// BODAS_RC18_12_40/Application/02 EasyConfig/DSM_easyConfig/Structure/DFC_bds_NoDeb0x80e2
{attribute 'external_name' := 'cmp_rts_DFC_bds_NoDeb0x80e2'}
TYPE DFC_bds_NoDeb0x80e2 : STRUCT
        DTC            : UDINT := 16#80E200;
        DFCid          : UINT  := 28;
        debounceMethod : USINT := TIME_IN_ROW;
    END_STRUCT
END_TYPE

// BODAS_RC18_12_40/Application/02 EasyConfig/DSM_easyConfig/Structure/DFC_bds_NoDeb0x80e3
{attribute 'external_name' := 'cmp_rts_DFC_bds_NoDeb0x80e3'}
TYPE DFC_bds_NoDeb0x80e3 : STRUCT
        DTC            : UDINT := 16#80E300;
        DFCid          : UINT  := 29;
        debounceMethod : USINT := TIME_IN_ROW;
    END_STRUCT
END_TYPE

// BODAS_RC18_12_40/Application/02 EasyConfig/DSM_easyConfig/Structure/DFC_bds_NoDeb0x80e4
{attribute 'external_name' := 'cmp_rts_DFC_bds_NoDeb0x80e4'}
TYPE DFC_bds_NoDeb0x80e4 : STRUCT
        DTC            : UDINT := 16#80E400;
        DFCid          : UINT  := 30;
        debounceMethod : USINT := TIME_IN_ROW;
    END_STRUCT
END_TYPE

// BODAS_RC18_12_40/Application/02 EasyConfig/DSM_easyConfig/Structure/DFC_bds_NoDeb0x80e5
{attribute 'external_name' := 'cmp_rts_DFC_bds_NoDeb0x80e5'}
TYPE DFC_bds_NoDeb0x80e5 : STRUCT
        DTC            : UDINT := 16#80E500;
        DFCid          : UINT  := 31;
        debounceMethod : USINT := TIME_IN_ROW;
    END_STRUCT
END_TYPE

// BODAS_RC18_12_40/Application/02 EasyConfig/DSM_easyConfig/Structure/DFC_bds_NoDeb0x80e6
{attribute 'external_name' := 'cmp_rts_DFC_bds_NoDeb0x80e6'}
TYPE DFC_bds_NoDeb0x80e6 : STRUCT
        DTC            : UDINT := 16#80E600;
        DFCid          : UINT  := 32;
        debounceMethod : USINT := TIME_IN_ROW;
    END_STRUCT
END_TYPE

// BODAS_RC18_12_40/Application/02 EasyConfig/DSM_easyConfig/Structure/DFC_bds_NoDeb0x80e7
{attribute 'external_name' := 'cmp_rts_DFC_bds_NoDeb0x80e7'}
TYPE DFC_bds_NoDeb0x80e7 : STRUCT
        DTC            : UDINT := 16#80E700;
        DFCid          : UINT  := 33;
        debounceMethod : USINT := TIME_IN_ROW;
    END_STRUCT
END_TYPE

// BODAS_RC18_12_40/Application/02 EasyConfig/DSM_easyConfig/Structure/DFC_bds_NoDeb0x80e8
{attribute 'external_name' := 'cmp_rts_DFC_bds_NoDeb0x80e8'}
TYPE DFC_bds_NoDeb0x80e8 : STRUCT
        DTC            : UDINT := 16#80E800;
        DFCid          : UINT  := 34;
        debounceMethod : USINT := TIME_IN_ROW;
    END_STRUCT
END_TYPE

// BODAS_RC18_12_40/Application/02 EasyConfig/DSM_easyConfig/Structure/DFC_bds_NoDeb0x80e9
{attribute 'external_name' := 'cmp_rts_DFC_bds_NoDeb0x80e9'}
TYPE DFC_bds_NoDeb0x80e9 : STRUCT
        DTC            : UDINT := 16#80E900;
        DFCid          : UINT  := 35;
        debounceMethod : USINT := TIME_IN_ROW;
    END_STRUCT
END_TYPE

// BODAS_RC18_12_40/Application/02 EasyConfig/DSM_easyConfig/Structure/DFC_bds_NoDeb0x80ea
{attribute 'external_name' := 'cmp_rts_DFC_bds_NoDeb0x80ea'}
TYPE DFC_bds_NoDeb0x80ea : STRUCT
        DTC            : UDINT := 16#80EA00;
        DFCid          : UINT  := 36;
        debounceMethod : USINT := TIME_IN_ROW;
    END_STRUCT
END_TYPE

// BODAS_RC18_12_40/Application/02 EasyConfig/DSM_easyConfig/Structure/DFC_bds_NoDeb0x80eb
{attribute 'external_name' := 'cmp_rts_DFC_bds_NoDeb0x80eb'}
TYPE DFC_bds_NoDeb0x80eb : STRUCT
        DTC            : UDINT := 16#80EB00;
        DFCid          : UINT  := 37;
        debounceMethod : USINT := TIME_IN_ROW;
    END_STRUCT
END_TYPE

// BODAS_RC18_12_40/Application/02 EasyConfig/DSM_easyConfig/Structure/DFC_bds_NoDeb0x80ec
{attribute 'external_name' := 'cmp_rts_DFC_bds_NoDeb0x80ec'}
TYPE DFC_bds_NoDeb0x80ec : STRUCT
        DTC            : UDINT := 16#80EC00;
        DFCid          : UINT  := 38;
        debounceMethod : USINT := TIME_IN_ROW;
    END_STRUCT
END_TYPE

// BODAS_RC18_12_40/Application/02 EasyConfig/DSM_easyConfig/Structure/DFC_bds_NoDeb0x80ed
{attribute 'external_name' := 'cmp_rts_DFC_bds_NoDeb0x80ed'}
TYPE DFC_bds_NoDeb0x80ed : STRUCT
        DTC            : UDINT := 16#80ED00;
        DFCid          : UINT  := 39;
        debounceMethod : USINT := TIME_IN_ROW;
    END_STRUCT
END_TYPE

// BODAS_RC18_12_40/Application/02 EasyConfig/DSM_easyConfig/Structure/DFC_bds_NoDeb0x80ee
{attribute 'external_name' := 'cmp_rts_DFC_bds_NoDeb0x80ee'}
TYPE DFC_bds_NoDeb0x80ee : STRUCT
        DTC            : UDINT := 16#80EE00;
        DFCid          : UINT  := 40;
        debounceMethod : USINT := TIME_IN_ROW;
    END_STRUCT
END_TYPE

// BODAS_RC18_12_40/Application/02 EasyConfig/DSM_easyConfig/Structure/DFC_bds_NoDeb0x80ef
{attribute 'external_name' := 'cmp_rts_DFC_bds_NoDeb0x80ef'}
TYPE DFC_bds_NoDeb0x80ef : STRUCT
        DTC            : UDINT := 16#80EF00;
        DFCid          : UINT  := 41;
        debounceMethod : USINT := TIME_IN_ROW;
    END_STRUCT
END_TYPE

// BODAS_RC18_12_40/Application/02 EasyConfig/DSM_easyConfig/Structure/DFC_bds_NoDeb0x80f0
{attribute 'external_name' := 'cmp_rts_DFC_bds_NoDeb0x80f0'}
TYPE DFC_bds_NoDeb0x80f0 : STRUCT
        DTC            : UDINT := 16#80F000;
        DFCid          : UINT  := 42;
        debounceMethod : USINT := TIME_IN_ROW;
    END_STRUCT
END_TYPE

// BODAS_RC18_12_40/Application/02 EasyConfig/DSM_easyConfig/Structure/DFC_bds_NoDeb0x80f1
{attribute 'external_name' := 'cmp_rts_DFC_bds_NoDeb0x80f1'}
TYPE DFC_bds_NoDeb0x80f1 : STRUCT
        DTC            : UDINT := 16#80F100;
        DFCid          : UINT  := 43;
        debounceMethod : USINT := TIME_IN_ROW;
    END_STRUCT
END_TYPE

// BODAS_RC18_12_40/Application/02 EasyConfig/DSM_easyConfig/Structure/DFC_bds_NoDeb0x80f2
{attribute 'external_name' := 'cmp_rts_DFC_bds_NoDeb0x80f2'}
TYPE DFC_bds_NoDeb0x80f2 : STRUCT
        DTC            : UDINT := 16#80F200;
        DFCid          : UINT  := 44;
        debounceMethod : USINT := TIME_IN_ROW;
    END_STRUCT
END_TYPE

// BODAS_RC18_12_40/Application/02 EasyConfig/DSM_easyConfig/Structure/DFC_bds_NoDeb0x80f3
{attribute 'external_name' := 'cmp_rts_DFC_bds_NoDeb0x80f3'}
TYPE DFC_bds_NoDeb0x80f3 : STRUCT
        DTC            : UDINT := 16#80F300;
        DFCid          : UINT  := 45;
        debounceMethod : USINT := TIME_IN_ROW;
    END_STRUCT
END_TYPE

// BODAS_RC18_12_40/Application/02 EasyConfig/DSM_easyConfig/Structure/DFC_bds_NoDeb0x80f4
{attribute 'external_name' := 'cmp_rts_DFC_bds_NoDeb0x80f4'}
TYPE DFC_bds_NoDeb0x80f4 : STRUCT
        DTC            : UDINT := 16#80F400;
        DFCid          : UINT  := 46;
        debounceMethod : USINT := TIME_IN_ROW;
    END_STRUCT
END_TYPE

// BODAS_RC18_12_40/Application/02 EasyConfig/DSM_easyConfig/Structure/DFC_bds_NoDeb0x80f5
{attribute 'external_name' := 'cmp_rts_DFC_bds_NoDeb0x80f5'}
TYPE DFC_bds_NoDeb0x80f5 : STRUCT
        DTC            : UDINT := 16#80F500;
        DFCid          : UINT  := 47;
        debounceMethod : USINT := TIME_IN_ROW;
    END_STRUCT
END_TYPE

// BODAS_RC18_12_40/Application/02 EasyConfig/DSM_easyConfig/Structure/DFC_bds_NoDeb0x80f6
{attribute 'external_name' := 'cmp_rts_DFC_bds_NoDeb0x80f6'}
TYPE DFC_bds_NoDeb0x80f6 : STRUCT
        DTC            : UDINT := 16#80F600;
        DFCid          : UINT  := 48;
        debounceMethod : USINT := TIME_IN_ROW;
    END_STRUCT
END_TYPE

// BODAS_RC18_12_40/Application/02 EasyConfig/DSM_easyConfig/Structure/DFC_bds_NoDeb0x80f7
{attribute 'external_name' := 'cmp_rts_DFC_bds_NoDeb0x80f7'}
TYPE DFC_bds_NoDeb0x80f7 : STRUCT
        DTC            : UDINT := 16#80F700;
        DFCid          : UINT  := 49;
        debounceMethod : USINT := TIME_IN_ROW;
    END_STRUCT
END_TYPE

// BODAS_RC18_12_40/Application/02 EasyConfig/DSM_easyConfig/Structure/DFC_bds_NoDeb0x80f8
{attribute 'external_name' := 'cmp_rts_DFC_bds_NoDeb0x80f8'}
TYPE DFC_bds_NoDeb0x80f8 : STRUCT
        DTC            : UDINT := 16#80F800;
        DFCid          : UINT  := 50;
        debounceMethod : USINT := TIME_IN_ROW;
    END_STRUCT
END_TYPE

// BODAS_RC18_12_40/Application/02 EasyConfig/DSM_easyConfig/Structure/DFC_bds_NoDeb0x80f9
{attribute 'external_name' := 'cmp_rts_DFC_bds_NoDeb0x80f9'}
TYPE DFC_bds_NoDeb0x80f9 : STRUCT
        DTC            : UDINT := 16#80F900;
        DFCid          : UINT  := 51;
        debounceMethod : USINT := TIME_IN_ROW;
    END_STRUCT
END_TYPE

// BODAS_RC18_12_40/Application/02 EasyConfig/DSM_easyConfig/Structure/DFC_bds_NoDeb0x80fa
{attribute 'external_name' := 'cmp_rts_DFC_bds_NoDeb0x80fa'}
TYPE DFC_bds_NoDeb0x80fa : STRUCT
        DTC            : UDINT := 16#80FA00;
        DFCid          : UINT  := 52;
        debounceMethod : USINT := TIME_IN_ROW;
    END_STRUCT
END_TYPE

// BODAS_RC18_12_40/Application/02 EasyConfig/DSM_easyConfig/Structure/DFC_bds_NoDeb0x80fb
{attribute 'external_name' := 'cmp_rts_DFC_bds_NoDeb0x80fb'}
TYPE DFC_bds_NoDeb0x80fb : STRUCT
        DTC            : UDINT := 16#80FB00;
        DFCid          : UINT  := 53;
        debounceMethod : USINT := TIME_IN_ROW;
    END_STRUCT
END_TYPE

// BODAS_RC18_12_40/Application/02 EasyConfig/DSM_easyConfig/Structure/DFC_bds_NoDeb0x80fc
{attribute 'external_name' := 'cmp_rts_DFC_bds_NoDeb0x80fc'}
TYPE DFC_bds_NoDeb0x80fc : STRUCT
        DTC            : UDINT := 16#80FC00;
        DFCid          : UINT  := 54;
        debounceMethod : USINT := TIME_IN_ROW;
    END_STRUCT
END_TYPE

// BODAS_RC18_12_40/Application/02 EasyConfig/DSM_easyConfig/Structure/DFC_bds_NoDeb0x80fd
{attribute 'external_name' := 'cmp_rts_DFC_bds_NoDeb0x80fd'}
TYPE DFC_bds_NoDeb0x80fd : STRUCT
        DTC            : UDINT := 16#80FD00;
        DFCid          : UINT  := 55;
        debounceMethod : USINT := TIME_IN_ROW;
    END_STRUCT
END_TYPE

// BODAS_RC18_12_40/Application/02 EasyConfig/DSM_easyConfig/Structure/DFC_bds_NoDeb0x80fe
{attribute 'external_name' := 'cmp_rts_DFC_bds_NoDeb0x80fe'}
TYPE DFC_bds_NoDeb0x80fe : STRUCT
        DTC            : UDINT := 16#80FE00;
        DFCid          : UINT  := 56;
        debounceMethod : USINT := TIME_IN_ROW;
    END_STRUCT
END_TYPE

// BODAS_RC18_12_40/Application/02 EasyConfig/DSM_easyConfig/Structure/DFC_bds_NoDeb0x80ff
{attribute 'external_name' := 'cmp_rts_DFC_bds_NoDeb0x80ff'}
TYPE DFC_bds_NoDeb0x80ff : STRUCT
        DTC            : UDINT := 16#80FF00;
        DFCid          : UINT  := 57;
        debounceMethod : USINT := TIME_IN_ROW;
    END_STRUCT
END_TYPE

// BODAS_RC18_12_40/Application/02 EasyConfig/DSM_easyConfig/Structure/DFC_bds_NoDeb0x8100
{attribute 'external_name' := 'cmp_rts_DFC_bds_NoDeb0x8100'}
TYPE DFC_bds_NoDeb0x8100 : STRUCT
        DTC            : UDINT := 16#810000;
        DFCid          : UINT  := 58;
        debounceMethod : USINT := TIME_IN_ROW;
    END_STRUCT
END_TYPE

// BODAS_RC18_12_40/Application/02 EasyConfig/DSM_easyConfig/Structure/DFC_bds_NoDeb0x8101
{attribute 'external_name' := 'cmp_rts_DFC_bds_NoDeb0x8101'}
TYPE DFC_bds_NoDeb0x8101 : STRUCT
        DTC            : UDINT := 16#810100;
        DFCid          : UINT  := 59;
        debounceMethod : USINT := TIME_IN_ROW;
    END_STRUCT
END_TYPE

// BODAS_RC18_12_40/Application/02 EasyConfig/DSM_easyConfig/Structure/DFC_bds_NoDeb0x8102
{attribute 'external_name' := 'cmp_rts_DFC_bds_NoDeb0x8102'}
TYPE DFC_bds_NoDeb0x8102 : STRUCT
        DTC            : UDINT := 16#810200;
        DFCid          : UINT  := 60;
        debounceMethod : USINT := TIME_IN_ROW;
    END_STRUCT
END_TYPE

// BODAS_RC18_12_40/Application/02 EasyConfig/DSM_easyConfig/Structure/DFC_bds_NoDeb0x8103
{attribute 'external_name' := 'cmp_rts_DFC_bds_NoDeb0x8103'}
TYPE DFC_bds_NoDeb0x8103 : STRUCT
        DTC            : UDINT := 16#810300;
        DFCid          : UINT  := 61;
        debounceMethod : USINT := TIME_IN_ROW;
    END_STRUCT
END_TYPE

// BODAS_RC18_12_40/Application/02 EasyConfig/DSM_easyConfig/Structure/DFC_bds_NoDeb0x8104
{attribute 'external_name' := 'cmp_rts_DFC_bds_NoDeb0x8104'}
TYPE DFC_bds_NoDeb0x8104 : STRUCT
        DTC            : UDINT := 16#810400;
        DFCid          : UINT  := 62;
        debounceMethod : USINT := TIME_IN_ROW;
    END_STRUCT
END_TYPE

// BODAS_RC18_12_40/Application/02 EasyConfig/DSM_easyConfig/Structure/DFC_bds_NoDeb0x8105
{attribute 'external_name' := 'cmp_rts_DFC_bds_NoDeb0x8105'}
TYPE DFC_bds_NoDeb0x8105 : STRUCT
        DTC            : UDINT := 16#810500;
        DFCid          : UINT  := 63;
        debounceMethod : USINT := TIME_IN_ROW;
    END_STRUCT
END_TYPE

// BODAS_RC18_12_40/Application/02 EasyConfig/DSM_easyConfig/Structure/DFC_bds_NoDeb0x8106
{attribute 'external_name' := 'cmp_rts_DFC_bds_NoDeb0x8106'}
TYPE DFC_bds_NoDeb0x8106 : STRUCT
        DTC            : UDINT := 16#810600;
        DFCid          : UINT  := 64;
        debounceMethod : USINT := TIME_IN_ROW;
    END_STRUCT
END_TYPE

// BODAS_RC18_12_40/Application/02 EasyConfig/DSM_easyConfig/Structure/DFC_bds_NoDeb0x8107
{attribute 'external_name' := 'cmp_rts_DFC_bds_NoDeb0x8107'}
TYPE DFC_bds_NoDeb0x8107 : STRUCT
        DTC            : UDINT := 16#810700;
        DFCid          : UINT  := 65;
        debounceMethod : USINT := TIME_IN_ROW;
    END_STRUCT
END_TYPE

// BODAS_RC18_12_40/Application/02 EasyConfig/DSM_easyConfig/Structure/DFC_bds_NoDeb0x8108
{attribute 'external_name' := 'cmp_rts_DFC_bds_NoDeb0x8108'}
TYPE DFC_bds_NoDeb0x8108 : STRUCT
        DTC            : UDINT := 16#810800;
        DFCid          : UINT  := 66;
        debounceMethod : USINT := TIME_IN_ROW;
    END_STRUCT
END_TYPE

// BODAS_RC18_12_40/Application/02 EasyConfig/DSM_easyConfig/Structure/DFC_bds_NoDeb0x8109
{attribute 'external_name' := 'cmp_rts_DFC_bds_NoDeb0x8109'}
TYPE DFC_bds_NoDeb0x8109 : STRUCT
        DTC            : UDINT := 16#810900;
        DFCid          : UINT  := 67;
        debounceMethod : USINT := TIME_IN_ROW;
    END_STRUCT
END_TYPE

// BODAS_RC18_12_40/Application/02 EasyConfig/DSM_easyConfig/Structure/DFC_bds_NoDeb0x810a
{attribute 'external_name' := 'cmp_rts_DFC_bds_NoDeb0x810a'}
TYPE DFC_bds_NoDeb0x810a : STRUCT
        DTC            : UDINT := 16#810A00;
        DFCid          : UINT  := 68;
        debounceMethod : USINT := TIME_IN_ROW;
    END_STRUCT
END_TYPE

// BODAS_RC18_12_40/Application/02 EasyConfig/DSM_easyConfig/Structure/DFC_bds_NoDeb0x810b
{attribute 'external_name' := 'cmp_rts_DFC_bds_NoDeb0x810b'}
TYPE DFC_bds_NoDeb0x810b : STRUCT
        DTC            : UDINT := 16#810B00;
        DFCid          : UINT  := 69;
        debounceMethod : USINT := TIME_IN_ROW;
    END_STRUCT
END_TYPE

// BODAS_RC18_12_40/Application/02 EasyConfig/DSM_easyConfig/Structure/DFC_bds_NoDeb0x810c
{attribute 'external_name' := 'cmp_rts_DFC_bds_NoDeb0x810c'}
TYPE DFC_bds_NoDeb0x810c : STRUCT
        DTC            : UDINT := 16#810C00;
        DFCid          : UINT  := 70;
        debounceMethod : USINT := TIME_IN_ROW;
    END_STRUCT
END_TYPE

// BODAS_RC18_12_40/Application/02 EasyConfig/DSM_easyConfig/Structure/DFC_bds_NoDeb0x810d
{attribute 'external_name' := 'cmp_rts_DFC_bds_NoDeb0x810d'}
TYPE DFC_bds_NoDeb0x810d : STRUCT
        DTC            : UDINT := 16#810D00;
        DFCid          : UINT  := 71;
        debounceMethod : USINT := TIME_IN_ROW;
    END_STRUCT
END_TYPE

// BODAS_RC18_12_40/Application/02 EasyConfig/DSM_easyConfig/Structure/DFC_bds_NoDeb0x810e
{attribute 'external_name' := 'cmp_rts_DFC_bds_NoDeb0x810e'}
TYPE DFC_bds_NoDeb0x810e : STRUCT
        DTC            : UDINT := 16#810E00;
        DFCid          : UINT  := 72;
        debounceMethod : USINT := TIME_IN_ROW;
    END_STRUCT
END_TYPE

// BODAS_RC18_12_40/Application/02 EasyConfig/DSM_easyConfig/Structure/DFC_bds_NoDeb0x810f
{attribute 'external_name' := 'cmp_rts_DFC_bds_NoDeb0x810f'}
TYPE DFC_bds_NoDeb0x810f : STRUCT
        DTC            : UDINT := 16#810F00;
        DFCid          : UINT  := 73;
        debounceMethod : USINT := TIME_IN_ROW;
    END_STRUCT
END_TYPE

// BODAS_RC18_12_40/Application/02 EasyConfig/DSM_easyConfig/Structure/DFC_bds_NoDeb0x8110
{attribute 'external_name' := 'cmp_rts_DFC_bds_NoDeb0x8110'}
TYPE DFC_bds_NoDeb0x8110 : STRUCT
        DTC            : UDINT := 16#811000;
        DFCid          : UINT  := 74;
        debounceMethod : USINT := TIME_IN_ROW;
    END_STRUCT
END_TYPE

// BODAS_RC18_12_40/Application/02 EasyConfig/DSM_easyConfig/Structure/DFC_bds_NoDeb0x8111
{attribute 'external_name' := 'cmp_rts_DFC_bds_NoDeb0x8111'}
TYPE DFC_bds_NoDeb0x8111 : STRUCT
        DTC            : UDINT := 16#811100;
        DFCid          : UINT  := 75;
        debounceMethod : USINT := TIME_IN_ROW;
    END_STRUCT
END_TYPE

// BODAS_RC18_12_40/Application/02 EasyConfig/DSM_easyConfig/Structure/DFC_bds_NoDeb0x8112
{attribute 'external_name' := 'cmp_rts_DFC_bds_NoDeb0x8112'}
TYPE DFC_bds_NoDeb0x8112 : STRUCT
        DTC            : UDINT := 16#811200;
        DFCid          : UINT  := 76;
        debounceMethod : USINT := TIME_IN_ROW;
    END_STRUCT
END_TYPE

// BODAS_RC18_12_40/Application/02 EasyConfig/DSM_easyConfig/Structure/DFC_bds_NoDeb0x8113
{attribute 'external_name' := 'cmp_rts_DFC_bds_NoDeb0x8113'}
TYPE DFC_bds_NoDeb0x8113 : STRUCT
        DTC            : UDINT := 16#811300;
        DFCid          : UINT  := 77;
        debounceMethod : USINT := TIME_IN_ROW;
    END_STRUCT
END_TYPE

// BODAS_RC18_12_40/Application/02 EasyConfig/DSM_easyConfig/Structure/DFC_bds_NoDeb0x8114
{attribute 'external_name' := 'cmp_rts_DFC_bds_NoDeb0x8114'}
TYPE DFC_bds_NoDeb0x8114 : STRUCT
        DTC            : UDINT := 16#811400;
        DFCid          : UINT  := 78;
        debounceMethod : USINT := TIME_IN_ROW;
    END_STRUCT
END_TYPE

// BODAS_RC18_12_40/Application/02 EasyConfig/DSM_easyConfig/Structure/DFC_bds_NoDeb0x8115
{attribute 'external_name' := 'cmp_rts_DFC_bds_NoDeb0x8115'}
TYPE DFC_bds_NoDeb0x8115 : STRUCT
        DTC            : UDINT := 16#811500;
        DFCid          : UINT  := 79;
        debounceMethod : USINT := TIME_IN_ROW;
    END_STRUCT
END_TYPE

// BODAS_RC18_12_40/Application/02 EasyConfig/DSM_easyConfig/Structure/DFC_bds_NoDeb0x8116
{attribute 'external_name' := 'cmp_rts_DFC_bds_NoDeb0x8116'}
TYPE DFC_bds_NoDeb0x8116 : STRUCT
        DTC            : UDINT := 16#811600;
        DFCid          : UINT  := 80;
        debounceMethod : USINT := TIME_IN_ROW;
    END_STRUCT
END_TYPE

// BODAS_RC18_12_40/Application/02 EasyConfig/DSM_easyConfig/Structure/DFC_bds_NoDeb0x8117
{attribute 'external_name' := 'cmp_rts_DFC_bds_NoDeb0x8117'}
TYPE DFC_bds_NoDeb0x8117 : STRUCT
        DTC            : UDINT := 16#811700;
        DFCid          : UINT  := 81;
        debounceMethod : USINT := TIME_IN_ROW;
    END_STRUCT
END_TYPE

// BODAS_RC18_12_40/Application/02 EasyConfig/DSM_easyConfig/Structure/DFC_bds_NoDeb0x8118
{attribute 'external_name' := 'cmp_rts_DFC_bds_NoDeb0x8118'}
TYPE DFC_bds_NoDeb0x8118 : STRUCT
        DTC            : UDINT := 16#811800;
        DFCid          : UINT  := 82;
        debounceMethod : USINT := TIME_IN_ROW;
    END_STRUCT
END_TYPE

// BODAS_RC18_12_40/Application/02 EasyConfig/DSM_easyConfig/Structure/DFC_bds_NoDeb0x8119
{attribute 'external_name' := 'cmp_rts_DFC_bds_NoDeb0x8119'}
TYPE DFC_bds_NoDeb0x8119 : STRUCT
        DTC            : UDINT := 16#811900;
        DFCid          : UINT  := 83;
        debounceMethod : USINT := TIME_IN_ROW;
    END_STRUCT
END_TYPE

// BODAS_RC18_12_40/Application/02 EasyConfig/DSM_easyConfig/Structure/DFC_bds_NoDeb0x811a
{attribute 'external_name' := 'cmp_rts_DFC_bds_NoDeb0x811a'}
TYPE DFC_bds_NoDeb0x811a : STRUCT
        DTC            : UDINT := 16#811A00;
        DFCid          : UINT  := 84;
        debounceMethod : USINT := TIME_IN_ROW;
    END_STRUCT
END_TYPE

// BODAS_RC18_12_40/Application/02 EasyConfig/DSM_easyConfig/Structure/DFC_bds_NoDeb0x811b
{attribute 'external_name' := 'cmp_rts_DFC_bds_NoDeb0x811b'}
TYPE DFC_bds_NoDeb0x811b : STRUCT
        DTC            : UDINT := 16#811B00;
        DFCid          : UINT  := 85;
        debounceMethod : USINT := TIME_IN_ROW;
    END_STRUCT
END_TYPE

// BODAS_RC18_12_40/Application/02 EasyConfig/DSM_easyConfig/Structure/DFC_bds_NoDeb0x811c
{attribute 'external_name' := 'cmp_rts_DFC_bds_NoDeb0x811c'}
TYPE DFC_bds_NoDeb0x811c : STRUCT
        DTC            : UDINT := 16#811C00;
        DFCid          : UINT  := 86;
        debounceMethod : USINT := TIME_IN_ROW;
    END_STRUCT
END_TYPE

// BODAS_RC18_12_40/Application/02 EasyConfig/DSM_easyConfig/Structure/DFC_bds_NoDeb0x811d
{attribute 'external_name' := 'cmp_rts_DFC_bds_NoDeb0x811d'}
TYPE DFC_bds_NoDeb0x811d : STRUCT
        DTC            : UDINT := 16#811D00;
        DFCid          : UINT  := 87;
        debounceMethod : USINT := TIME_IN_ROW;
    END_STRUCT
END_TYPE

// BODAS_RC18_12_40/Application/02 EasyConfig/DSM_easyConfig/Structure/DFC_bds_NoDeb0x811e
{attribute 'external_name' := 'cmp_rts_DFC_bds_NoDeb0x811e'}
TYPE DFC_bds_NoDeb0x811e : STRUCT
        DTC            : UDINT := 16#811E00;
        DFCid          : UINT  := 88;
        debounceMethod : USINT := TIME_IN_ROW;
    END_STRUCT
END_TYPE

// BODAS_RC18_12_40/Application/02 EasyConfig/DSM_easyConfig/Structure/DFC_bds_NoDeb0x811f
{attribute 'external_name' := 'cmp_rts_DFC_bds_NoDeb0x811f'}
TYPE DFC_bds_NoDeb0x811f : STRUCT
        DTC            : UDINT := 16#811F00;
        DFCid          : UINT  := 89;
        debounceMethod : USINT := TIME_IN_ROW;
    END_STRUCT
END_TYPE

// BODAS_RC18_12_40/Application/02 EasyConfig/DSM_easyConfig/Structure/DFC_bds_NoDeb0x8120
{attribute 'external_name' := 'cmp_rts_DFC_bds_NoDeb0x8120'}
TYPE DFC_bds_NoDeb0x8120 : STRUCT
        DTC            : UDINT := 16#812000;
        DFCid          : UINT  := 90;
        debounceMethod : USINT := TIME_IN_ROW;
    END_STRUCT
END_TYPE

// BODAS_RC18_12_40/Application/02 EasyConfig/DSM_easyConfig/Structure/DFC_bds_NoDeb0x8121
{attribute 'external_name' := 'cmp_rts_DFC_bds_NoDeb0x8121'}
TYPE DFC_bds_NoDeb0x8121 : STRUCT
        DTC            : UDINT := 16#812100;
        DFCid          : UINT  := 91;
        debounceMethod : USINT := TIME_IN_ROW;
    END_STRUCT
END_TYPE

// BODAS_RC18_12_40/Application/02 EasyConfig/DSM_easyConfig/Structure/DFC_bds_NoDeb0x8122
{attribute 'external_name' := 'cmp_rts_DFC_bds_NoDeb0x8122'}
TYPE DFC_bds_NoDeb0x8122 : STRUCT
        DTC            : UDINT := 16#812200;
        DFCid          : UINT  := 92;
        debounceMethod : USINT := TIME_IN_ROW;
    END_STRUCT
END_TYPE

// BODAS_RC18_12_40/Application/02 EasyConfig/DSM_easyConfig/Structure/DFC_bds_NoDeb0x8123
{attribute 'external_name' := 'cmp_rts_DFC_bds_NoDeb0x8123'}
TYPE DFC_bds_NoDeb0x8123 : STRUCT
        DTC            : UDINT := 16#812300;
        DFCid          : UINT  := 93;
        debounceMethod : USINT := TIME_IN_ROW;
    END_STRUCT
END_TYPE

// BODAS_RC18_12_40/Application/02 EasyConfig/DSM_easyConfig/Structure/DFC_bds_NoDeb0x8124
{attribute 'external_name' := 'cmp_rts_DFC_bds_NoDeb0x8124'}
TYPE DFC_bds_NoDeb0x8124 : STRUCT
        DTC            : UDINT := 16#812400;
        DFCid          : UINT  := 94;
        debounceMethod : USINT := TIME_IN_ROW;
    END_STRUCT
END_TYPE

// BODAS_RC18_12_40/Application/02 EasyConfig/DSM_easyConfig/Structure/DFC_bds_NoDeb0x8125
{attribute 'external_name' := 'cmp_rts_DFC_bds_NoDeb0x8125'}
TYPE DFC_bds_NoDeb0x8125 : STRUCT
        DTC            : UDINT := 16#812500;
        DFCid          : UINT  := 95;
        debounceMethod : USINT := TIME_IN_ROW;
    END_STRUCT
END_TYPE

// BODAS_RC18_12_40/Application/02 EasyConfig/DSM_easyConfig/Structure/DFC_bds_NoDeb0x8126
{attribute 'external_name' := 'cmp_rts_DFC_bds_NoDeb0x8126'}
TYPE DFC_bds_NoDeb0x8126 : STRUCT
        DTC            : UDINT := 16#812600;
        DFCid          : UINT  := 96;
        debounceMethod : USINT := TIME_IN_ROW;
    END_STRUCT
END_TYPE

// BODAS_RC18_12_40/Application/02 EasyConfig/DSM_easyConfig/Structure/DFC_bds_NoDeb0x8127
{attribute 'external_name' := 'cmp_rts_DFC_bds_NoDeb0x8127'}
TYPE DFC_bds_NoDeb0x8127 : STRUCT
        DTC            : UDINT := 16#812700;
        DFCid          : UINT  := 97;
        debounceMethod : USINT := TIME_IN_ROW;
    END_STRUCT
END_TYPE

// BODAS_RC18_12_40/Application/02 EasyConfig/DSM_easyConfig/Structure/DFC_bds_NoDeb0x8128
{attribute 'external_name' := 'cmp_rts_DFC_bds_NoDeb0x8128'}
TYPE DFC_bds_NoDeb0x8128 : STRUCT
        DTC            : UDINT := 16#812800;
        DFCid          : UINT  := 98;
        debounceMethod : USINT := TIME_IN_ROW;
    END_STRUCT
END_TYPE

// BODAS_RC18_12_40/Application/02 EasyConfig/DSM_easyConfig/Structure/DFC_bds_NoDeb0x8129
{attribute 'external_name' := 'cmp_rts_DFC_bds_NoDeb0x8129'}
TYPE DFC_bds_NoDeb0x8129 : STRUCT
        DTC            : UDINT := 16#812900;
        DFCid          : UINT  := 99;
        debounceMethod : USINT := TIME_IN_ROW;
    END_STRUCT
END_TYPE

// BODAS_RC18_12_40/Application/02 EasyConfig/DSM_easyConfig/Structure/DFC_bds_NoDeb0x812a
{attribute 'external_name' := 'cmp_rts_DFC_bds_NoDeb0x812a'}
TYPE DFC_bds_NoDeb0x812a : STRUCT
        DTC            : UDINT := 16#812A00;
        DFCid          : UINT  := 100;
        debounceMethod : USINT := TIME_IN_ROW;
    END_STRUCT
END_TYPE

// BODAS_RC18_12_40/Application/02 EasyConfig/DSM_easyConfig/Structure/DFC_bds_NoDeb0x8C01
{attribute 'external_name' := 'cmp_rts_DFC_bds_NoDeb0x8C01'}
TYPE DFC_bds_NoDeb0x8C01 : STRUCT
        DTC            : UDINT := 16#8C0100;
        DFCid          : UINT  := 820;
        debounceMethod : USINT := NO_DEBOUNCE;
    END_STRUCT
END_TYPE

// BODAS_RC18_12_40/Application/02 EasyConfig/DSM_easyConfig/Structure/DFC_bds_NoDeb0x8C02
{attribute 'external_name' := 'cmp_rts_DFC_bds_NoDeb0x8C02'}
TYPE DFC_bds_NoDeb0x8C02 : STRUCT
        DTC            : UDINT := 16#8C0200;
        DFCid          : UINT  := 821;
        debounceMethod : USINT := NO_DEBOUNCE;
    END_STRUCT
END_TYPE

// BODAS_RC18_12_40/Application/02 EasyConfig/DSM_easyConfig/Structure/DFC_bds_NoDeb0x8C03
{attribute 'external_name' := 'cmp_rts_DFC_bds_NoDeb0x8C03'}
TYPE DFC_bds_NoDeb0x8C03 : STRUCT
        DTC            : UDINT := 16#8C0300;
        DFCid          : UINT  := 822;
        debounceMethod : USINT := NO_DEBOUNCE;
    END_STRUCT
END_TYPE

// BODAS_RC18_12_40/Application/02 EasyConfig/DSM_easyConfig/Structure/DFC_bds_TiInRow0x8B01
{attribute 'external_name' := 'cmp_rts_DFC_bds_TiInRow0x8B01'}
TYPE DFC_bds_TiInRow0x8B01 : STRUCT
        DTC            : UDINT := 16#8B0100;
        DFCid          : UINT  := 101;
        debounceMethod : USINT := TIME_IN_ROW;
    END_STRUCT
END_TYPE

// BODAS_RC18_12_40/Application/02 EasyConfig/DSM_easyConfig/Structure/DFC_bds_TiInRow0x8B02
{attribute 'external_name' := 'cmp_rts_DFC_bds_TiInRow0x8B02'}
TYPE DFC_bds_TiInRow0x8B02 : STRUCT
        DTC            : UDINT := 16#8B0200;
        DFCid          : UINT  := 102;
        debounceMethod : USINT := TIME_IN_ROW;
    END_STRUCT
END_TYPE

// BODAS_RC18_12_40/Application/02 EasyConfig/DSM_easyConfig/Structure/DFC_bds_TiInRow0x8B03
{attribute 'external_name' := 'cmp_rts_DFC_bds_TiInRow0x8B03'}
TYPE DFC_bds_TiInRow0x8B03 : STRUCT
        DTC            : UDINT := 16#8B0300;
        DFCid          : UINT  := 103;
        debounceMethod : USINT := TIME_IN_ROW;
    END_STRUCT
END_TYPE

// BODAS_RC18_12_40/Application/02 EasyConfig/DSM_easyConfig/Structure/DFC_bds_TiUpDwn0x8A01
{attribute 'external_name' := 'cmp_rts_DFC_bds_TiUpDwn0x8A01'}
TYPE DFC_bds_TiUpDwn0x8A01 : STRUCT
        DTC            : UDINT := 16#8A0100;
        DFCid          : UINT  := 206;
        debounceMethod : USINT := TIME_UP_DOWN;
    END_STRUCT
END_TYPE

// BODAS_RC18_12_40/Application/02 EasyConfig/DSM_easyConfig/Structure/DFC_bds_TiUpDwn0x8A02
{attribute 'external_name' := 'cmp_rts_DFC_bds_TiUpDwn0x8A02'}
TYPE DFC_bds_TiUpDwn0x8A02 : STRUCT
        DTC            : UDINT := 16#8A0200;
        DFCid          : UINT  := 207;
        debounceMethod : USINT := TIME_UP_DOWN;
    END_STRUCT
END_TYPE

// BODAS_RC18_12_40/Application/02 EasyConfig/DSM_easyConfig/Structure/DFC_bds_TiUpDwn0x8A03
{attribute 'external_name' := 'cmp_rts_DFC_bds_TiUpDwn0x8A03'}
TYPE DFC_bds_TiUpDwn0x8A03 : STRUCT
        DTC            : UDINT := 16#8A0300;
        DFCid          : UINT  := 208;
        debounceMethod : USINT := TIME_UP_DOWN;
    END_STRUCT
END_TYPE

// BODAS_RC18_12_40/Application/02 EasyConfig/DSM_easyConfig/Structure/DFC_CAN_E_TIMEOUT
{attribute 'external_name' := 'cmp_rts_DFC_CAN_E_TIMEOUT'}
TYPE DFC_CAN_E_TIMEOUT : STRUCT
        DTC            : UDINT := 16#094200;
        DFCid          : UINT  := 1165;
        debounceMethod : USINT := NO_DEBOUNCE;
    END_STRUCT
END_TYPE

// BODAS_RC18_12_40/Application/02 EasyConfig/DSM_easyConfig/Structure/DFC_CANSM_E_BUS_OFF_NETWORK_0
{attribute 'external_name' := 'cmp_rts_DFC_CANSM_E_BUS_OFF_NETWORK_0'}
TYPE DFC_CANSM_E_BUS_OFF_NETWORK_0 : STRUCT
        DTC            : UDINT := 16#104C00;
        DFCid          : UINT  := 1160;
        debounceMethod : USINT := NO_DEBOUNCE;
    END_STRUCT
END_TYPE

// BODAS_RC18_12_40/Application/02 EasyConfig/DSM_easyConfig/Structure/DFC_CANSM_E_BUS_OFF_NETWORK_1
{attribute 'external_name' := 'cmp_rts_DFC_CANSM_E_BUS_OFF_NETWORK_1'}
TYPE DFC_CANSM_E_BUS_OFF_NETWORK_1 : STRUCT
        DTC            : UDINT := 16#104D00;
        DFCid          : UINT  := 1161;
        debounceMethod : USINT := NO_DEBOUNCE;
    END_STRUCT
END_TYPE

// BODAS_RC18_12_40/Application/02 EasyConfig/DSM_easyConfig/Structure/DFC_CANSM_E_BUS_OFF_NETWORK_2
{attribute 'external_name' := 'cmp_rts_DFC_CANSM_E_BUS_OFF_NETWORK_2'}
TYPE DFC_CANSM_E_BUS_OFF_NETWORK_2 : STRUCT
        DTC            : UDINT := 16#104E00;
        DFCid          : UINT  := 1162;
        debounceMethod : USINT := NO_DEBOUNCE;
    END_STRUCT
END_TYPE

// BODAS_RC18_12_40/Application/02 EasyConfig/DSM_easyConfig/Structure/DFC_CANSM_E_BUS_OFF_NETWORK_3
{attribute 'external_name' := 'cmp_rts_DFC_CANSM_E_BUS_OFF_NETWORK_3'}
TYPE DFC_CANSM_E_BUS_OFF_NETWORK_3 : STRUCT
        DTC            : UDINT := 16#104F00;
        DFCid          : UINT  := 1163;
        debounceMethod : USINT := NO_DEBOUNCE;
    END_STRUCT
END_TYPE

// BODAS_RC18_12_40/Application/02 EasyConfig/DSM_easyConfig/Structure/DFC_CANTRCV_E_NO_TRCV_CONTROL_0
{attribute 'external_name' := 'cmp_rts_DFC_CANTRCV_E_NO_TRCV_CONTROL_0'}
TYPE DFC_CANTRCV_E_NO_TRCV_CONTROL_0 : STRUCT
        DTC            : UDINT := 16#094000;
        DFCid          : UINT  := 1164;
        debounceMethod : USINT := NO_DEBOUNCE;
    END_STRUCT
END_TYPE

// BODAS_RC18_12_40/Application/02 EasyConfig/DSM_easyConfig/Structure/DFC_Com_numWhlIncFrtLeft
{attribute 'external_name' := 'cmp_rts_DFC_Com_numWhlIncFrtLeft'}
TYPE DFC_Com_numWhlIncFrtLeft : STRUCT
        DTC : UDINT := 16#103A00;
    END_STRUCT
END_TYPE

// BODAS_RC18_12_40/Application/02 EasyConfig/DSM_easyConfig/Structure/DFC_Com_stWhlSensRrRht
{attribute 'external_name' := 'cmp_rts_DFC_Com_stWhlSensRrRht'}
TYPE DFC_Com_stWhlSensRrRht : STRUCT
        DTC : UDINT := 16#103B00;
    END_STRUCT
END_TYPE

// BODAS_RC18_12_40/Application/02 EasyConfig/DSM_easyConfig/Structure/DFC_Com_trqClthTCSDCSDes
{attribute 'external_name' := 'cmp_rts_DFC_Com_trqClthTCSDCSDes'}
TYPE DFC_Com_trqClthTCSDCSDes : STRUCT
        DTC : UDINT := 16#103C00;
    END_STRUCT
END_TYPE

// BODAS_RC18_12_40/Application/02 EasyConfig/DSM_easyConfig/Structure/DFC_Com_vWhlRrL
{attribute 'external_name' := 'cmp_rts_DFC_Com_vWhlRrL'}
TYPE DFC_Com_vWhlRrL : STRUCT
        DTC : UDINT := 16#103D00;
    END_STRUCT
END_TYPE

// BODAS_RC18_12_40/Application/02 EasyConfig/DSM_easyConfig/Structure/DFC_ComChksACC_06
{attribute 'external_name' := 'cmp_rts_DFC_ComChksACC_06'}
TYPE DFC_ComChksACC_06 : STRUCT
        DTC : UDINT := 16#101600;
    END_STRUCT
END_TYPE

// BODAS_RC18_12_40/Application/02 EasyConfig/DSM_easyConfig/Structure/DFC_ComChksBMS_01
{attribute 'external_name' := 'cmp_rts_DFC_ComChksBMS_01'}
TYPE DFC_ComChksBMS_01 : STRUCT
        DTC : UDINT := 16#101700;
    END_STRUCT
END_TYPE

// BODAS_RC18_12_40/Application/02 EasyConfig/DSM_easyConfig/Structure/DFC_ComChksESP_02
{attribute 'external_name' := 'cmp_rts_DFC_ComChksESP_02'}
TYPE DFC_ComChksESP_02 : STRUCT
        DTC : UDINT := 16#101800;
    END_STRUCT
END_TYPE

// BODAS_RC18_12_40/Application/02 EasyConfig/DSM_easyConfig/Structure/DFC_ComChksESP_05
{attribute 'external_name' := 'cmp_rts_DFC_ComChksESP_05'}
TYPE DFC_ComChksESP_05 : STRUCT
        DTC : UDINT := 16#101900;
    END_STRUCT
END_TYPE

// BODAS_RC18_12_40/Application/02 EasyConfig/DSM_easyConfig/Structure/DFC_ComChksESP_07
{attribute 'external_name' := 'cmp_rts_DFC_ComChksESP_07'}
TYPE DFC_ComChksESP_07 : STRUCT
        DTC : UDINT := 16#101A00;
    END_STRUCT
END_TYPE

// BODAS_RC18_12_40/Application/02 EasyConfig/DSM_easyConfig/Structure/DFC_ComChksESP_10
{attribute 'external_name' := 'cmp_rts_DFC_ComChksESP_10'}
TYPE DFC_ComChksESP_10 : STRUCT
        DTC : UDINT := 16#101B00;
    END_STRUCT
END_TYPE

// BODAS_RC18_12_40/Application/02 EasyConfig/DSM_easyConfig/Structure/DFC_ComChksESP_19
{attribute 'external_name' := 'cmp_rts_DFC_ComChksESP_19'}
TYPE DFC_ComChksESP_19 : STRUCT
        DTC : UDINT := 16#101C00;
    END_STRUCT
END_TYPE

// BODAS_RC18_12_40/Application/02 EasyConfig/DSM_easyConfig/Structure/DFC_ComChksESP_20
{attribute 'external_name' := 'cmp_rts_DFC_ComChksESP_20'}
TYPE DFC_ComChksESP_20 : STRUCT
        DTC : UDINT := 16#101D00;
    END_STRUCT
END_TYPE

// BODAS_RC18_12_40/Application/02 EasyConfig/DSM_easyConfig/Structure/DFC_ComChksESP_21
{attribute 'external_name' := 'cmp_rts_DFC_ComChksESP_21'}
TYPE DFC_ComChksESP_21 : STRUCT
        DTC : UDINT := 16#101E00;
    END_STRUCT
END_TYPE

// BODAS_RC18_12_40/Application/02 EasyConfig/DSM_easyConfig/Structure/DFC_ComChksKlemmen_Status_01
{attribute 'external_name' := 'cmp_rts_DFC_ComChksKlemmen_Status_01'}
TYPE DFC_ComChksKlemmen_Status_01 : STRUCT
        DTC : UDINT := 16#103800;
    END_STRUCT
END_TYPE

// BODAS_RC18_12_40/Application/02 EasyConfig/DSM_easyConfig/Structure/DFC_ComCntACC_06
{attribute 'external_name' := 'cmp_rts_DFC_ComCntACC_06'}
TYPE DFC_ComCntACC_06 : STRUCT
        DTC : UDINT := 16#101F00;
    END_STRUCT
END_TYPE

// BODAS_RC18_12_40/Application/02 EasyConfig/DSM_easyConfig/Structure/DFC_ComCntBMS_01
{attribute 'external_name' := 'cmp_rts_DFC_ComCntBMS_01'}
TYPE DFC_ComCntBMS_01 : STRUCT
        DTC : UDINT := 16#102000;
    END_STRUCT
END_TYPE

// BODAS_RC18_12_40/Application/02 EasyConfig/DSM_easyConfig/Structure/DFC_ComCntESP_02
{attribute 'external_name' := 'cmp_rts_DFC_ComCntESP_02'}
TYPE DFC_ComCntESP_02 : STRUCT
        DTC : UDINT := 16#102100;
    END_STRUCT
END_TYPE

// BODAS_RC18_12_40/Application/02 EasyConfig/DSM_easyConfig/Structure/DFC_ComCntESP_05
{attribute 'external_name' := 'cmp_rts_DFC_ComCntESP_05'}
TYPE DFC_ComCntESP_05 : STRUCT
        DTC : UDINT := 16#102200;
    END_STRUCT
END_TYPE

// BODAS_RC18_12_40/Application/02 EasyConfig/DSM_easyConfig/Structure/DFC_ComCntESP_07
{attribute 'external_name' := 'cmp_rts_DFC_ComCntESP_07'}
TYPE DFC_ComCntESP_07 : STRUCT
        DTC : UDINT := 16#102300;
    END_STRUCT
END_TYPE

// BODAS_RC18_12_40/Application/02 EasyConfig/DSM_easyConfig/Structure/DFC_ComCntESP_10
{attribute 'external_name' := 'cmp_rts_DFC_ComCntESP_10'}
TYPE DFC_ComCntESP_10 : STRUCT
        DTC : UDINT := 16#102400;
    END_STRUCT
END_TYPE

// BODAS_RC18_12_40/Application/02 EasyConfig/DSM_easyConfig/Structure/DFC_ComCntESP_19
{attribute 'external_name' := 'cmp_rts_DFC_ComCntESP_19'}
TYPE DFC_ComCntESP_19 : STRUCT
        DTC : UDINT := 16#102500;
    END_STRUCT
END_TYPE

// BODAS_RC18_12_40/Application/02 EasyConfig/DSM_easyConfig/Structure/DFC_ComCntESP_20
{attribute 'external_name' := 'cmp_rts_DFC_ComCntESP_20'}
TYPE DFC_ComCntESP_20 : STRUCT
        DTC : UDINT := 16#102600;
    END_STRUCT
END_TYPE

// BODAS_RC18_12_40/Application/02 EasyConfig/DSM_easyConfig/Structure/DFC_ComCntESP_21
{attribute 'external_name' := 'cmp_rts_DFC_ComCntESP_21'}
TYPE DFC_ComCntESP_21 : STRUCT
        DTC : UDINT := 16#102700;
    END_STRUCT
END_TYPE

// BODAS_RC18_12_40/Application/02 EasyConfig/DSM_easyConfig/Structure/DFC_ComCntKlemmen_Status_01
{attribute 'external_name' := 'cmp_rts_DFC_ComCntKlemmen_Status_01'}
TYPE DFC_ComCntKlemmen_Status_01 : STRUCT
        DTC : UDINT := 16#103900;
    END_STRUCT
END_TYPE

// BODAS_RC18_12_40/Application/02 EasyConfig/DSM_easyConfig/Structure/DFC_ComDlcACC_06
{attribute 'external_name' := 'cmp_rts_DFC_ComDlcACC_06'}
TYPE DFC_ComDlcACC_06 : STRUCT
        DTC : UDINT := 16#102800;
    END_STRUCT
END_TYPE

// BODAS_RC18_12_40/Application/02 EasyConfig/DSM_easyConfig/Structure/DFC_ComDlcESP_02
{attribute 'external_name' := 'cmp_rts_DFC_ComDlcESP_02'}
TYPE DFC_ComDlcESP_02 : STRUCT
        DTC : UDINT := 16#102900;
    END_STRUCT
END_TYPE

// BODAS_RC18_12_40/Application/02 EasyConfig/DSM_easyConfig/Structure/DFC_ComDlcESP_05
{attribute 'external_name' := 'cmp_rts_DFC_ComDlcESP_05'}
TYPE DFC_ComDlcESP_05 : STRUCT
        DTC : UDINT := 16#102A00;
    END_STRUCT
END_TYPE

// BODAS_RC18_12_40/Application/02 EasyConfig/DSM_easyConfig/Structure/DFC_ComDlcESP_07
{attribute 'external_name' := 'cmp_rts_DFC_ComDlcESP_07'}
TYPE DFC_ComDlcESP_07 : STRUCT
        DTC : UDINT := 16#102B00;
    END_STRUCT
END_TYPE

// BODAS_RC18_12_40/Application/02 EasyConfig/DSM_easyConfig/Structure/DFC_ComDlcESP_10
{attribute 'external_name' := 'cmp_rts_DFC_ComDlcESP_10'}
TYPE DFC_ComDlcESP_10 : STRUCT
        DTC : UDINT := 16#102C00;
    END_STRUCT
END_TYPE

// BODAS_RC18_12_40/Application/02 EasyConfig/DSM_easyConfig/Structure/DFC_ComDlcESP_19
{attribute 'external_name' := 'cmp_rts_DFC_ComDlcESP_19'}
TYPE DFC_ComDlcESP_19 : STRUCT
        DTC : UDINT := 16#102D00;
    END_STRUCT
END_TYPE

// BODAS_RC18_12_40/Application/02 EasyConfig/DSM_easyConfig/Structure/DFC_ComDlcESP_20
{attribute 'external_name' := 'cmp_rts_DFC_ComDlcESP_20'}
TYPE DFC_ComDlcESP_20 : STRUCT
        DTC : UDINT := 16#102E00;
    END_STRUCT
END_TYPE

// BODAS_RC18_12_40/Application/02 EasyConfig/DSM_easyConfig/Structure/DFC_ComDlcESP_21
{attribute 'external_name' := 'cmp_rts_DFC_ComDlcESP_21'}
TYPE DFC_ComDlcESP_21 : STRUCT
        DTC : UDINT := 16#102F00;
    END_STRUCT
END_TYPE

// BODAS_RC18_12_40/Application/02 EasyConfig/DSM_easyConfig/Structure/DFC_COMM_E_NET_START_IND_CHANNEL_0
{attribute 'external_name' := 'cmp_rts_DFC_COMM_E_NET_START_IND_CHANNEL_0'}
TYPE DFC_COMM_E_NET_START_IND_CHANNEL_0 : STRUCT
        DTC            : UDINT := 16#105000;
        DFCid          : UINT  := 1166;
        debounceMethod : USINT := NO_DEBOUNCE;
    END_STRUCT
END_TYPE

// BODAS_RC18_12_40/Application/02 EasyConfig/DSM_easyConfig/Structure/DFC_COMM_E_NET_START_IND_CHANNEL_1
{attribute 'external_name' := 'cmp_rts_DFC_COMM_E_NET_START_IND_CHANNEL_1'}
TYPE DFC_COMM_E_NET_START_IND_CHANNEL_1 : STRUCT
        DTC            : UDINT := 16#105100;
        DFCid          : UINT  := 1167;
        debounceMethod : USINT := NO_DEBOUNCE;
    END_STRUCT
END_TYPE

// BODAS_RC18_12_40/Application/02 EasyConfig/DSM_easyConfig/Structure/DFC_COMM_E_NET_START_IND_CHANNEL_2
{attribute 'external_name' := 'cmp_rts_DFC_COMM_E_NET_START_IND_CHANNEL_2'}
TYPE DFC_COMM_E_NET_START_IND_CHANNEL_2 : STRUCT
        DTC            : UDINT := 16#105200;
        DFCid          : UINT  := 1168;
        debounceMethod : USINT := NO_DEBOUNCE;
    END_STRUCT
END_TYPE

// BODAS_RC18_12_40/Application/02 EasyConfig/DSM_easyConfig/Structure/DFC_COMM_E_NET_START_IND_CHANNEL_3
{attribute 'external_name' := 'cmp_rts_DFC_COMM_E_NET_START_IND_CHANNEL_3'}
TYPE DFC_COMM_E_NET_START_IND_CHANNEL_3 : STRUCT
        DTC            : UDINT := 16#105300;
        DFCid          : UINT  := 1169;
        debounceMethod : USINT := NO_DEBOUNCE;
    END_STRUCT
END_TYPE

// BODAS_RC18_12_40/Application/02 EasyConfig/DSM_easyConfig/Structure/DFC_COMM_E_NET_START_IND_CHANNEL_4
{attribute 'external_name' := 'cmp_rts_DFC_COMM_E_NET_START_IND_CHANNEL_4'}
TYPE DFC_COMM_E_NET_START_IND_CHANNEL_4 : STRUCT
        DTC            : UDINT := 16#105400;
        DFCid          : UINT  := 1170;
        debounceMethod : USINT := NO_DEBOUNCE;
    END_STRUCT
END_TYPE

// BODAS_RC18_12_40/Application/02 EasyConfig/DSM_easyConfig/Structure/DFC_COMM_E_NET_START_IND_CHANNEL_5
{attribute 'external_name' := 'cmp_rts_DFC_COMM_E_NET_START_IND_CHANNEL_5'}
TYPE DFC_COMM_E_NET_START_IND_CHANNEL_5 : STRUCT
        DTC            : UDINT := 16#105500;
        DFCid          : UINT  := 1171;
        debounceMethod : USINT := NO_DEBOUNCE;
    END_STRUCT
END_TYPE

// BODAS_RC18_12_40/Application/02 EasyConfig/DSM_easyConfig/Structure/DFC_ComTOutACC_06
{attribute 'external_name' := 'cmp_rts_DFC_ComTOutACC_06'}
TYPE DFC_ComTOutACC_06 : STRUCT
        DTC : UDINT := 16#103000;
    END_STRUCT
END_TYPE

// BODAS_RC18_12_40/Application/02 EasyConfig/DSM_easyConfig/Structure/DFC_ComTOutESP_02
{attribute 'external_name' := 'cmp_rts_DFC_ComTOutESP_02'}
TYPE DFC_ComTOutESP_02 : STRUCT
        DTC : UDINT := 16#103100;
    END_STRUCT
END_TYPE

// BODAS_RC18_12_40/Application/02 EasyConfig/DSM_easyConfig/Structure/DFC_ComTOutESP_05
{attribute 'external_name' := 'cmp_rts_DFC_ComTOutESP_05'}
TYPE DFC_ComTOutESP_05 : STRUCT
        DTC : UDINT := 16#103200;
    END_STRUCT
END_TYPE

// BODAS_RC18_12_40/Application/02 EasyConfig/DSM_easyConfig/Structure/DFC_ComTOutESP_07
{attribute 'external_name' := 'cmp_rts_DFC_ComTOutESP_07'}
TYPE DFC_ComTOutESP_07 : STRUCT
        DTC : UDINT := 16#103300;
    END_STRUCT
END_TYPE

// BODAS_RC18_12_40/Application/02 EasyConfig/DSM_easyConfig/Structure/DFC_ComTOutESP_10
{attribute 'external_name' := 'cmp_rts_DFC_ComTOutESP_10'}
TYPE DFC_ComTOutESP_10 : STRUCT
        DTC : UDINT := 16#103400;
    END_STRUCT
END_TYPE

// BODAS_RC18_12_40/Application/02 EasyConfig/DSM_easyConfig/Structure/DFC_ComTOutESP_19
{attribute 'external_name' := 'cmp_rts_DFC_ComTOutESP_19'}
TYPE DFC_ComTOutESP_19 : STRUCT
        DTC : UDINT := 16#103500;
    END_STRUCT
END_TYPE

// BODAS_RC18_12_40/Application/02 EasyConfig/DSM_easyConfig/Structure/DFC_ComTOutESP_20
{attribute 'external_name' := 'cmp_rts_DFC_ComTOutESP_20'}
TYPE DFC_ComTOutESP_20 : STRUCT
        DTC : UDINT := 16#103600;
    END_STRUCT
END_TYPE

// BODAS_RC18_12_40/Application/02 EasyConfig/DSM_easyConfig/Structure/DFC_ComTOutESP_21
{attribute 'external_name' := 'cmp_rts_DFC_ComTOutESP_21'}
TYPE DFC_ComTOutESP_21 : STRUCT
        DTC : UDINT := 16#103700;
    END_STRUCT
END_TYPE

// BODAS_RC18_12_40/Application/02 EasyConfig/DSM_easyConfig/Structure/DFC_DevLibBattUHi
{attribute 'external_name' := 'cmp_rts_DFC_DevLibBattUHi'}
TYPE DFC_DevLibBattUHi : STRUCT
        DTC            : UDINT := 16#092300;
        DFCid          : UINT  := 104;
        debounceMethod : USINT := TIME_UP_DOWN;
    END_STRUCT
END_TYPE

// BODAS_RC18_12_40/Application/02 EasyConfig/DSM_easyConfig/Structure/DFC_DevLibBattULo
{attribute 'external_name' := 'cmp_rts_DFC_DevLibBattULo'}
TYPE DFC_DevLibBattULo : STRUCT
        DTC            : UDINT := 16#092400;
        DFCid          : UINT  := 105;
        debounceMethod : USINT := TIME_UP_DOWN;
    END_STRUCT
END_TYPE

// BODAS_RC18_12_40/Application/02 EasyConfig/DSM_easyConfig/Structure/DFC_DSMDummy
{attribute 'external_name' := 'cmp_rts_DFC_DSMDummy'}
TYPE DFC_DSMDummy : STRUCT
        DTC            : UDINT := 16#100F00;
        DFCid          : UINT  := 720;
        debounceMethod : USINT := NO_DEBOUNCE;
    END_STRUCT
END_TYPE

// BODAS_RC18_12_40/Application/02 EasyConfig/DSM_easyConfig/Structure/DFC_LIN_E_TIMEOUT
{attribute 'external_name' := 'cmp_rts_DFC_LIN_E_TIMEOUT'}
TYPE DFC_LIN_E_TIMEOUT : STRUCT
        DTC            : UDINT := 16#094100;
        DFCid          : UINT  := 1172;
        debounceMethod : USINT := NO_DEBOUNCE;
    END_STRUCT
END_TYPE

// BODAS_RC18_12_40/Application/02 EasyConfig/DSM_easyConfig/Structure/DFC_MoCSOPICO
{attribute 'external_name' := 'cmp_rts_DFC_MoCSOPICO'}
TYPE DFC_MoCSOPICO : STRUCT
        DTC            : UDINT := 16#106000;
        DFCid          : UINT  := 1296;
        debounceMethod : USINT := NATIVE;
    END_STRUCT
END_TYPE

// BODAS_RC18_12_40/Application/02 EasyConfig/DSM_easyConfig/Structure/DFC_MoFVarPostBldSel
{attribute 'external_name' := 'cmp_rts_DFC_MoFVarPostBldSel'}
TYPE DFC_MoFVarPostBldSel : STRUCT
        DTC            : UDINT := 16#098900;
        DFCid          : UINT  := 1297;
        debounceMethod : USINT := NATIVE;
    END_STRUCT
END_TYPE

// BODAS_RC18_12_40/Application/02 EasyConfig/DSM_easyConfig/Structure/DFC_MoSysCtrlReIni
{attribute 'external_name' := 'cmp_rts_DFC_MoSysCtrlReIni'}
TYPE DFC_MoSysCtrlReIni : STRUCT
        DTC            : UDINT := 16#106100;
        DFCid          : UINT  := 1298;
        debounceMethod : USINT := NATIVE;
    END_STRUCT
END_TYPE

// BODAS_RC18_12_40/Application/02 EasyConfig/DSM_easyConfig/Structure/DFC_MOXEMM_SMU_ALM0_0
{attribute 'external_name' := 'cmp_rts_DFC_MOXEMM_SMU_ALM0_0'}
TYPE DFC_MOXEMM_SMU_ALM0_0 : STRUCT
        DTC            : UDINT := 16#106200;
        DFCid          : UINT  := 1185;
        debounceMethod : USINT := NATIVE;
    END_STRUCT
END_TYPE

// BODAS_RC18_12_40/Application/02 EasyConfig/DSM_easyConfig/Structure/DFC_MOXEMM_SMU_ALM0_10
{attribute 'external_name' := 'cmp_rts_DFC_MOXEMM_SMU_ALM0_10'}
TYPE DFC_MOXEMM_SMU_ALM0_10 : STRUCT
        DTC            : UDINT := 16#106900;
        DFCid          : UINT  := 1187;
        debounceMethod : USINT := NATIVE;
    END_STRUCT
END_TYPE

// BODAS_RC18_12_40/Application/02 EasyConfig/DSM_easyConfig/Structure/DFC_MOXEMM_SMU_ALM0_11
{attribute 'external_name' := 'cmp_rts_DFC_MOXEMM_SMU_ALM0_11'}
TYPE DFC_MOXEMM_SMU_ALM0_11 : STRUCT
        DTC            : UDINT := 16#106A00;
        DFCid          : UINT  := 1188;
        debounceMethod : USINT := NATIVE;
    END_STRUCT
END_TYPE

// BODAS_RC18_12_40/Application/02 EasyConfig/DSM_easyConfig/Structure/DFC_MOXEMM_SMU_ALM0_13
{attribute 'external_name' := 'cmp_rts_DFC_MOXEMM_SMU_ALM0_13'}
TYPE DFC_MOXEMM_SMU_ALM0_13 : STRUCT
        DTC            : UDINT := 16#106B00;
        DFCid          : UINT  := 1189;
        debounceMethod : USINT := NATIVE;
    END_STRUCT
END_TYPE

// BODAS_RC18_12_40/Application/02 EasyConfig/DSM_easyConfig/Structure/DFC_MOXEMM_SMU_ALM0_14
{attribute 'external_name' := 'cmp_rts_DFC_MOXEMM_SMU_ALM0_14'}
TYPE DFC_MOXEMM_SMU_ALM0_14 : STRUCT
        DTC            : UDINT := 16#106C00;
        DFCid          : UINT  := 1190;
        debounceMethod : USINT := NATIVE;
    END_STRUCT
END_TYPE

// BODAS_RC18_12_40/Application/02 EasyConfig/DSM_easyConfig/Structure/DFC_MOXEMM_SMU_ALM0_1
{attribute 'external_name' := 'cmp_rts_DFC_MOXEMM_SMU_ALM0_1'}
TYPE DFC_MOXEMM_SMU_ALM0_1 : STRUCT
        DTC            : UDINT := 16#106300;
        DFCid          : UINT  := 1186;
        debounceMethod : USINT := NATIVE;
    END_STRUCT
END_TYPE

// BODAS_RC18_12_40/Application/02 EasyConfig/DSM_easyConfig/Structure/DFC_MOXEMM_SMU_ALM0_22
{attribute 'external_name' := 'cmp_rts_DFC_MOXEMM_SMU_ALM0_22'}
TYPE DFC_MOXEMM_SMU_ALM0_22 : STRUCT
        DTC            : UDINT := 16#106D00;
        DFCid          : UINT  := 1192;
        debounceMethod : USINT := NATIVE;
    END_STRUCT
END_TYPE

// BODAS_RC18_12_40/Application/02 EasyConfig/DSM_easyConfig/Structure/DFC_MOXEMM_SMU_ALM0_23
{attribute 'external_name' := 'cmp_rts_DFC_MOXEMM_SMU_ALM0_23'}
TYPE DFC_MOXEMM_SMU_ALM0_23 : STRUCT
        DTC            : UDINT := 16#106E00;
        DFCid          : UINT  := 1193;
        debounceMethod : USINT := NATIVE;
    END_STRUCT
END_TYPE

// BODAS_RC18_12_40/Application/02 EasyConfig/DSM_easyConfig/Structure/DFC_MOXEMM_SMU_ALM0_2
{attribute 'external_name' := 'cmp_rts_DFC_MOXEMM_SMU_ALM0_2'}
TYPE DFC_MOXEMM_SMU_ALM0_2 : STRUCT
        DTC            : UDINT := 16#106400;
        DFCid          : UINT  := 1191;
        debounceMethod : USINT := NATIVE;
    END_STRUCT
END_TYPE

// BODAS_RC18_12_40/Application/02 EasyConfig/DSM_easyConfig/Structure/DFC_MOXEMM_SMU_ALM0_4
{attribute 'external_name' := 'cmp_rts_DFC_MOXEMM_SMU_ALM0_4'}
TYPE DFC_MOXEMM_SMU_ALM0_4 : STRUCT
        DTC            : UDINT := 16#106500;
        DFCid          : UINT  := 1194;
        debounceMethod : USINT := NATIVE;
    END_STRUCT
END_TYPE

// BODAS_RC18_12_40/Application/02 EasyConfig/DSM_easyConfig/Structure/DFC_MOXEMM_SMU_ALM0_5
{attribute 'external_name' := 'cmp_rts_DFC_MOXEMM_SMU_ALM0_5'}
TYPE DFC_MOXEMM_SMU_ALM0_5 : STRUCT
        DTC            : UDINT := 16#106600;
        DFCid          : UINT  := 1195;
        debounceMethod : USINT := NATIVE;
    END_STRUCT
END_TYPE

// BODAS_RC18_12_40/Application/02 EasyConfig/DSM_easyConfig/Structure/DFC_MOXEMM_SMU_ALM0_7
{attribute 'external_name' := 'cmp_rts_DFC_MOXEMM_SMU_ALM0_7'}
TYPE DFC_MOXEMM_SMU_ALM0_7 : STRUCT
        DTC            : UDINT := 16#106700;
        DFCid          : UINT  := 1196;
        debounceMethod : USINT := NATIVE;
    END_STRUCT
END_TYPE

// BODAS_RC18_12_40/Application/02 EasyConfig/DSM_easyConfig/Structure/DFC_MOXEMM_SMU_ALM0_8
{attribute 'external_name' := 'cmp_rts_DFC_MOXEMM_SMU_ALM0_8'}
TYPE DFC_MOXEMM_SMU_ALM0_8 : STRUCT
        DTC            : UDINT := 16#106800;
        DFCid          : UINT  := 1197;
        debounceMethod : USINT := NATIVE;
    END_STRUCT
END_TYPE

// BODAS_RC18_12_40/Application/02 EasyConfig/DSM_easyConfig/Structure/DFC_MOXEMM_SMU_ALM10_16
{attribute 'external_name' := 'cmp_rts_DFC_MOXEMM_SMU_ALM10_16'}
TYPE DFC_MOXEMM_SMU_ALM10_16 : STRUCT
        DTC            : UDINT := 16#10C200;
        DFCid          : UINT  := 1198;
        debounceMethod : USINT := NATIVE;
    END_STRUCT
END_TYPE

// BODAS_RC18_12_40/Application/02 EasyConfig/DSM_easyConfig/Structure/DFC_MOXEMM_SMU_ALM10_17
{attribute 'external_name' := 'cmp_rts_DFC_MOXEMM_SMU_ALM10_17'}
TYPE DFC_MOXEMM_SMU_ALM10_17 : STRUCT
        DTC            : UDINT := 16#10C300;
        DFCid          : UINT  := 1199;
        debounceMethod : USINT := NATIVE;
    END_STRUCT
END_TYPE

// BODAS_RC18_12_40/Application/02 EasyConfig/DSM_easyConfig/Structure/DFC_MOXEMM_SMU_ALM10_21
{attribute 'external_name' := 'cmp_rts_DFC_MOXEMM_SMU_ALM10_21'}
TYPE DFC_MOXEMM_SMU_ALM10_21 : STRUCT
        DTC            : UDINT := 16#10C400;
        DFCid          : UINT  := 1200;
        debounceMethod : USINT := NATIVE;
    END_STRUCT
END_TYPE

// BODAS_RC18_12_40/Application/02 EasyConfig/DSM_easyConfig/Structure/DFC_MOXEMM_SMU_ALM11_0
{attribute 'external_name' := 'cmp_rts_DFC_MOXEMM_SMU_ALM11_0'}
TYPE DFC_MOXEMM_SMU_ALM11_0 : STRUCT
        DTC            : UDINT := 16#10C500;
        DFCid          : UINT  := 1201;
        debounceMethod : USINT := NATIVE;
    END_STRUCT
END_TYPE

// BODAS_RC18_12_40/Application/02 EasyConfig/DSM_easyConfig/Structure/DFC_MOXEMM_SMU_ALM11_1
{attribute 'external_name' := 'cmp_rts_DFC_MOXEMM_SMU_ALM11_1'}
TYPE DFC_MOXEMM_SMU_ALM11_1 : STRUCT
        DTC            : UDINT := 16#10C600;
        DFCid          : UINT  := 1202;
        debounceMethod : USINT := NATIVE;
    END_STRUCT
END_TYPE

// BODAS_RC18_12_40/Application/02 EasyConfig/DSM_easyConfig/Structure/DFC_MOXEMM_SMU_ALM11_2
{attribute 'external_name' := 'cmp_rts_DFC_MOXEMM_SMU_ALM11_2'}
TYPE DFC_MOXEMM_SMU_ALM11_2 : STRUCT
        DTC            : UDINT := 16#10C700;
        DFCid          : UINT  := 1203;
        debounceMethod : USINT := NATIVE;
    END_STRUCT
END_TYPE

// BODAS_RC18_12_40/Application/02 EasyConfig/DSM_easyConfig/Structure/DFC_MOXEMM_SMU_ALM11_3
{attribute 'external_name' := 'cmp_rts_DFC_MOXEMM_SMU_ALM11_3'}
TYPE DFC_MOXEMM_SMU_ALM11_3 : STRUCT
        DTC            : UDINT := 16#10C800;
        DFCid          : UINT  := 1204;
        debounceMethod : USINT := NATIVE;
    END_STRUCT
END_TYPE

// BODAS_RC18_12_40/Application/02 EasyConfig/DSM_easyConfig/Structure/DFC_MOXEMM_SMU_ALM11_4
{attribute 'external_name' := 'cmp_rts_DFC_MOXEMM_SMU_ALM11_4'}
TYPE DFC_MOXEMM_SMU_ALM11_4 : STRUCT
        DTC            : UDINT := 16#10C900;
        DFCid          : UINT  := 1205;
        debounceMethod : USINT := NATIVE;
    END_STRUCT
END_TYPE

// BODAS_RC18_12_40/Application/02 EasyConfig/DSM_easyConfig/Structure/DFC_MOXEMM_SMU_ALM11_5
{attribute 'external_name' := 'cmp_rts_DFC_MOXEMM_SMU_ALM11_5'}
TYPE DFC_MOXEMM_SMU_ALM11_5 : STRUCT
        DTC            : UDINT := 16#10CA00;
        DFCid          : UINT  := 1206;
        debounceMethod : USINT := NATIVE;
    END_STRUCT
END_TYPE

// BODAS_RC18_12_40/Application/02 EasyConfig/DSM_easyConfig/Structure/DFC_MOXEMM_SMU_ALM11_8
{attribute 'external_name' := 'cmp_rts_DFC_MOXEMM_SMU_ALM11_8'}
TYPE DFC_MOXEMM_SMU_ALM11_8 : STRUCT
        DTC            : UDINT := 16#10CB00;
        DFCid          : UINT  := 1207;
        debounceMethod : USINT := NATIVE;
    END_STRUCT
END_TYPE

// BODAS_RC18_12_40/Application/02 EasyConfig/DSM_easyConfig/Structure/DFC_MOXEMM_SMU_ALM11_9
{attribute 'external_name' := 'cmp_rts_DFC_MOXEMM_SMU_ALM11_9'}
TYPE DFC_MOXEMM_SMU_ALM11_9 : STRUCT
        DTC            : UDINT := 16#10CC00;
        DFCid          : UINT  := 1208;
        debounceMethod : USINT := NATIVE;
    END_STRUCT
END_TYPE

// BODAS_RC18_12_40/Application/02 EasyConfig/DSM_easyConfig/Structure/DFC_MOXEMM_SMU_ALM1_0
{attribute 'external_name' := 'cmp_rts_DFC_MOXEMM_SMU_ALM1_0'}
TYPE DFC_MOXEMM_SMU_ALM1_0 : STRUCT
        DTC            : UDINT := 16#106F00;
        DFCid          : UINT  := 1209;
        debounceMethod : USINT := NATIVE;
    END_STRUCT
END_TYPE

// BODAS_RC18_12_40/Application/02 EasyConfig/DSM_easyConfig/Structure/DFC_MOXEMM_SMU_ALM1_10
{attribute 'external_name' := 'cmp_rts_DFC_MOXEMM_SMU_ALM1_10'}
TYPE DFC_MOXEMM_SMU_ALM1_10 : STRUCT
        DTC            : UDINT := 16#107600;
        DFCid          : UINT  := 1211;
        debounceMethod : USINT := NATIVE;
    END_STRUCT
END_TYPE

// BODAS_RC18_12_40/Application/02 EasyConfig/DSM_easyConfig/Structure/DFC_MOXEMM_SMU_ALM1_11
{attribute 'external_name' := 'cmp_rts_DFC_MOXEMM_SMU_ALM1_11'}
TYPE DFC_MOXEMM_SMU_ALM1_11 : STRUCT
        DTC            : UDINT := 16#107700;
        DFCid          : UINT  := 1212;
        debounceMethod : USINT := NATIVE;
    END_STRUCT
END_TYPE

// BODAS_RC18_12_40/Application/02 EasyConfig/DSM_easyConfig/Structure/DFC_MOXEMM_SMU_ALM1_13
{attribute 'external_name' := 'cmp_rts_DFC_MOXEMM_SMU_ALM1_13'}
TYPE DFC_MOXEMM_SMU_ALM1_13 : STRUCT
        DTC            : UDINT := 16#107800;
        DFCid          : UINT  := 1213;
        debounceMethod : USINT := NATIVE;
    END_STRUCT
END_TYPE

// BODAS_RC18_12_40/Application/02 EasyConfig/DSM_easyConfig/Structure/DFC_MOXEMM_SMU_ALM1_14
{attribute 'external_name' := 'cmp_rts_DFC_MOXEMM_SMU_ALM1_14'}
TYPE DFC_MOXEMM_SMU_ALM1_14 : STRUCT
        DTC            : UDINT := 16#107900;
        DFCid          : UINT  := 1214;
        debounceMethod : USINT := NATIVE;
    END_STRUCT
END_TYPE

// BODAS_RC18_12_40/Application/02 EasyConfig/DSM_easyConfig/Structure/DFC_MOXEMM_SMU_ALM1_1
{attribute 'external_name' := 'cmp_rts_DFC_MOXEMM_SMU_ALM1_1'}
TYPE DFC_MOXEMM_SMU_ALM1_1 : STRUCT
        DTC            : UDINT := 16#107000;
        DFCid          : UINT  := 1210;
        debounceMethod : USINT := NATIVE;
    END_STRUCT
END_TYPE

// BODAS_RC18_12_40/Application/02 EasyConfig/DSM_easyConfig/Structure/DFC_MOXEMM_SMU_ALM1_22
{attribute 'external_name' := 'cmp_rts_DFC_MOXEMM_SMU_ALM1_22'}
TYPE DFC_MOXEMM_SMU_ALM1_22 : STRUCT
        DTC            : UDINT := 16#107A00;
        DFCid          : UINT  := 1216;
        debounceMethod : USINT := NATIVE;
    END_STRUCT
END_TYPE

// BODAS_RC18_12_40/Application/02 EasyConfig/DSM_easyConfig/Structure/DFC_MOXEMM_SMU_ALM1_23
{attribute 'external_name' := 'cmp_rts_DFC_MOXEMM_SMU_ALM1_23'}
TYPE DFC_MOXEMM_SMU_ALM1_23 : STRUCT
        DTC            : UDINT := 16#107B00;
        DFCid          : UINT  := 1217;
        debounceMethod : USINT := NATIVE;
    END_STRUCT
END_TYPE

// BODAS_RC18_12_40/Application/02 EasyConfig/DSM_easyConfig/Structure/DFC_MOXEMM_SMU_ALM1_2
{attribute 'external_name' := 'cmp_rts_DFC_MOXEMM_SMU_ALM1_2'}
TYPE DFC_MOXEMM_SMU_ALM1_2 : STRUCT
        DTC            : UDINT := 16#107100;
        DFCid          : UINT  := 1215;
        debounceMethod : USINT := NATIVE;
    END_STRUCT
END_TYPE

// BODAS_RC18_12_40/Application/02 EasyConfig/DSM_easyConfig/Structure/DFC_MOXEMM_SMU_ALM1_4
{attribute 'external_name' := 'cmp_rts_DFC_MOXEMM_SMU_ALM1_4'}
TYPE DFC_MOXEMM_SMU_ALM1_4 : STRUCT
        DTC            : UDINT := 16#107200;
        DFCid          : UINT  := 1218;
        debounceMethod : USINT := NATIVE;
    END_STRUCT
END_TYPE

// BODAS_RC18_12_40/Application/02 EasyConfig/DSM_easyConfig/Structure/DFC_MOXEMM_SMU_ALM1_5
{attribute 'external_name' := 'cmp_rts_DFC_MOXEMM_SMU_ALM1_5'}
TYPE DFC_MOXEMM_SMU_ALM1_5 : STRUCT
        DTC            : UDINT := 16#107300;
        DFCid          : UINT  := 1219;
        debounceMethod : USINT := NATIVE;
    END_STRUCT
END_TYPE

// BODAS_RC18_12_40/Application/02 EasyConfig/DSM_easyConfig/Structure/DFC_MOXEMM_SMU_ALM1_7
{attribute 'external_name' := 'cmp_rts_DFC_MOXEMM_SMU_ALM1_7'}
TYPE DFC_MOXEMM_SMU_ALM1_7 : STRUCT
        DTC            : UDINT := 16#107400;
        DFCid          : UINT  := 1220;
        debounceMethod : USINT := NATIVE;
    END_STRUCT
END_TYPE

// BODAS_RC18_12_40/Application/02 EasyConfig/DSM_easyConfig/Structure/DFC_MOXEMM_SMU_ALM1_8
{attribute 'external_name' := 'cmp_rts_DFC_MOXEMM_SMU_ALM1_8'}
TYPE DFC_MOXEMM_SMU_ALM1_8 : STRUCT
        DTC            : UDINT := 16#107500;
        DFCid          : UINT  := 1221;
        debounceMethod : USINT := NATIVE;
    END_STRUCT
END_TYPE

// BODAS_RC18_12_40/Application/02 EasyConfig/DSM_easyConfig/Structure/DFC_MOXEMM_SMU_ALM21_0
{attribute 'external_name' := 'cmp_rts_DFC_MOXEMM_SMU_ALM21_0'}
TYPE DFC_MOXEMM_SMU_ALM21_0 : STRUCT
        DTC            : UDINT := 16#10CD00;
        DFCid          : UINT  := 1222;
        debounceMethod : USINT := NATIVE;
    END_STRUCT
END_TYPE

// BODAS_RC18_12_40/Application/02 EasyConfig/DSM_easyConfig/Structure/DFC_MOXEMM_SMU_ALM21_16
{attribute 'external_name' := 'cmp_rts_DFC_MOXEMM_SMU_ALM21_16'}
TYPE DFC_MOXEMM_SMU_ALM21_16 : STRUCT
        DTC            : UDINT := 16#10CF00;
        DFCid          : UINT  := 1223;
        debounceMethod : USINT := NATIVE;
    END_STRUCT
END_TYPE

// BODAS_RC18_12_40/Application/02 EasyConfig/DSM_easyConfig/Structure/DFC_MOXEMM_SMU_ALM21_3
{attribute 'external_name' := 'cmp_rts_DFC_MOXEMM_SMU_ALM21_3'}
TYPE DFC_MOXEMM_SMU_ALM21_3 : STRUCT
        DTC            : UDINT := 16#10CE00;
        DFCid          : UINT  := 1224;
        debounceMethod : USINT := NATIVE;
    END_STRUCT
END_TYPE

// BODAS_RC18_12_40/Application/02 EasyConfig/DSM_easyConfig/Structure/DFC_MOXEMM_SMU_ALM2_10
{attribute 'external_name' := 'cmp_rts_DFC_MOXEMM_SMU_ALM2_10'}
TYPE DFC_MOXEMM_SMU_ALM2_10 : STRUCT
        DTC            : UDINT := 16#108200;
        DFCid          : UINT  := 1226;
        debounceMethod : USINT := NATIVE;
    END_STRUCT
END_TYPE

// BODAS_RC18_12_40/Application/02 EasyConfig/DSM_easyConfig/Structure/DFC_MOXEMM_SMU_ALM2_11
{attribute 'external_name' := 'cmp_rts_DFC_MOXEMM_SMU_ALM2_11'}
TYPE DFC_MOXEMM_SMU_ALM2_11 : STRUCT
        DTC            : UDINT := 16#108300;
        DFCid          : UINT  := 1227;
        debounceMethod : USINT := NATIVE;
    END_STRUCT
END_TYPE

// BODAS_RC18_12_40/Application/02 EasyConfig/DSM_easyConfig/Structure/DFC_MOXEMM_SMU_ALM2_13
{attribute 'external_name' := 'cmp_rts_DFC_MOXEMM_SMU_ALM2_13'}
TYPE DFC_MOXEMM_SMU_ALM2_13 : STRUCT
        DTC            : UDINT := 16#108400;
        DFCid          : UINT  := 1228;
        debounceMethod : USINT := NATIVE;
    END_STRUCT
END_TYPE

// BODAS_RC18_12_40/Application/02 EasyConfig/DSM_easyConfig/Structure/DFC_MOXEMM_SMU_ALM2_14
{attribute 'external_name' := 'cmp_rts_DFC_MOXEMM_SMU_ALM2_14'}
TYPE DFC_MOXEMM_SMU_ALM2_14 : STRUCT
        DTC            : UDINT := 16#108500;
        DFCid          : UINT  := 1229;
        debounceMethod : USINT := NATIVE;
    END_STRUCT
END_TYPE

// BODAS_RC18_12_40/Application/02 EasyConfig/DSM_easyConfig/Structure/DFC_MOXEMM_SMU_ALM2_1
{attribute 'external_name' := 'cmp_rts_DFC_MOXEMM_SMU_ALM2_1'}
TYPE DFC_MOXEMM_SMU_ALM2_1 : STRUCT
        DTC            : UDINT := 16#107C00;
        DFCid          : UINT  := 1225;
        debounceMethod : USINT := NATIVE;
    END_STRUCT
END_TYPE

// BODAS_RC18_12_40/Application/02 EasyConfig/DSM_easyConfig/Structure/DFC_MOXEMM_SMU_ALM2_22
{attribute 'external_name' := 'cmp_rts_DFC_MOXEMM_SMU_ALM2_22'}
TYPE DFC_MOXEMM_SMU_ALM2_22 : STRUCT
        DTC            : UDINT := 16#108600;
        DFCid          : UINT  := 1231;
        debounceMethod : USINT := NATIVE;
    END_STRUCT
END_TYPE

// BODAS_RC18_12_40/Application/02 EasyConfig/DSM_easyConfig/Structure/DFC_MOXEMM_SMU_ALM2_23
{attribute 'external_name' := 'cmp_rts_DFC_MOXEMM_SMU_ALM2_23'}
TYPE DFC_MOXEMM_SMU_ALM2_23 : STRUCT
        DTC            : UDINT := 16#108700;
        DFCid          : UINT  := 1232;
        debounceMethod : USINT := NATIVE;
    END_STRUCT
END_TYPE

// BODAS_RC18_12_40/Application/02 EasyConfig/DSM_easyConfig/Structure/DFC_MOXEMM_SMU_ALM2_2
{attribute 'external_name' := 'cmp_rts_DFC_MOXEMM_SMU_ALM2_2'}
TYPE DFC_MOXEMM_SMU_ALM2_2 : STRUCT
        DTC            : UDINT := 16#107D00;
        DFCid          : UINT  := 1230;
        debounceMethod : USINT := NATIVE;
    END_STRUCT
END_TYPE

// BODAS_RC18_12_40/Application/02 EasyConfig/DSM_easyConfig/Structure/DFC_MOXEMM_SMU_ALM2_4
{attribute 'external_name' := 'cmp_rts_DFC_MOXEMM_SMU_ALM2_4'}
TYPE DFC_MOXEMM_SMU_ALM2_4 : STRUCT
        DTC            : UDINT := 16#107E00;
        DFCid          : UINT  := 1233;
        debounceMethod : USINT := NATIVE;
    END_STRUCT
END_TYPE

// BODAS_RC18_12_40/Application/02 EasyConfig/DSM_easyConfig/Structure/DFC_MOXEMM_SMU_ALM2_5
{attribute 'external_name' := 'cmp_rts_DFC_MOXEMM_SMU_ALM2_5'}
TYPE DFC_MOXEMM_SMU_ALM2_5 : STRUCT
        DTC            : UDINT := 16#107F00;
        DFCid          : UINT  := 1234;
        debounceMethod : USINT := NATIVE;
    END_STRUCT
END_TYPE

// BODAS_RC18_12_40/Application/02 EasyConfig/DSM_easyConfig/Structure/DFC_MOXEMM_SMU_ALM2_7
{attribute 'external_name' := 'cmp_rts_DFC_MOXEMM_SMU_ALM2_7'}
TYPE DFC_MOXEMM_SMU_ALM2_7 : STRUCT
        DTC            : UDINT := 16#108000;
        DFCid          : UINT  := 1235;
        debounceMethod : USINT := NATIVE;
    END_STRUCT
END_TYPE

// BODAS_RC18_12_40/Application/02 EasyConfig/DSM_easyConfig/Structure/DFC_MOXEMM_SMU_ALM2_8
{attribute 'external_name' := 'cmp_rts_DFC_MOXEMM_SMU_ALM2_8'}
TYPE DFC_MOXEMM_SMU_ALM2_8 : STRUCT
        DTC            : UDINT := 16#108100;
        DFCid          : UINT  := 1236;
        debounceMethod : USINT := NATIVE;
    END_STRUCT
END_TYPE

// BODAS_RC18_12_40/Application/02 EasyConfig/DSM_easyConfig/Structure/DFC_MOXEMM_SMU_ALM3_10
{attribute 'external_name' := 'cmp_rts_DFC_MOXEMM_SMU_ALM3_10'}
TYPE DFC_MOXEMM_SMU_ALM3_10 : STRUCT
        DTC            : UDINT := 16#108E00;
        DFCid          : UINT  := 1238;
        debounceMethod : USINT := NATIVE;
    END_STRUCT
END_TYPE

// BODAS_RC18_12_40/Application/02 EasyConfig/DSM_easyConfig/Structure/DFC_MOXEMM_SMU_ALM3_11
{attribute 'external_name' := 'cmp_rts_DFC_MOXEMM_SMU_ALM3_11'}
TYPE DFC_MOXEMM_SMU_ALM3_11 : STRUCT
        DTC            : UDINT := 16#108F00;
        DFCid          : UINT  := 1239;
        debounceMethod : USINT := NATIVE;
    END_STRUCT
END_TYPE

// BODAS_RC18_12_40/Application/02 EasyConfig/DSM_easyConfig/Structure/DFC_MOXEMM_SMU_ALM3_13
{attribute 'external_name' := 'cmp_rts_DFC_MOXEMM_SMU_ALM3_13'}
TYPE DFC_MOXEMM_SMU_ALM3_13 : STRUCT
        DTC            : UDINT := 16#109000;
        DFCid          : UINT  := 1240;
        debounceMethod : USINT := NATIVE;
    END_STRUCT
END_TYPE

// BODAS_RC18_12_40/Application/02 EasyConfig/DSM_easyConfig/Structure/DFC_MOXEMM_SMU_ALM3_14
{attribute 'external_name' := 'cmp_rts_DFC_MOXEMM_SMU_ALM3_14'}
TYPE DFC_MOXEMM_SMU_ALM3_14 : STRUCT
        DTC            : UDINT := 16#109100;
        DFCid          : UINT  := 1241;
        debounceMethod : USINT := NATIVE;
    END_STRUCT
END_TYPE

// BODAS_RC18_12_40/Application/02 EasyConfig/DSM_easyConfig/Structure/DFC_MOXEMM_SMU_ALM3_1
{attribute 'external_name' := 'cmp_rts_DFC_MOXEMM_SMU_ALM3_1'}
TYPE DFC_MOXEMM_SMU_ALM3_1 : STRUCT
        DTC            : UDINT := 16#108800;
        DFCid          : UINT  := 1237;
        debounceMethod : USINT := NATIVE;
    END_STRUCT
END_TYPE

// BODAS_RC18_12_40/Application/02 EasyConfig/DSM_easyConfig/Structure/DFC_MOXEMM_SMU_ALM3_22
{attribute 'external_name' := 'cmp_rts_DFC_MOXEMM_SMU_ALM3_22'}
TYPE DFC_MOXEMM_SMU_ALM3_22 : STRUCT
        DTC            : UDINT := 16#109200;
        DFCid          : UINT  := 1243;
        debounceMethod : USINT := NATIVE;
    END_STRUCT
END_TYPE

// BODAS_RC18_12_40/Application/02 EasyConfig/DSM_easyConfig/Structure/DFC_MOXEMM_SMU_ALM3_23
{attribute 'external_name' := 'cmp_rts_DFC_MOXEMM_SMU_ALM3_23'}
TYPE DFC_MOXEMM_SMU_ALM3_23 : STRUCT
        DTC            : UDINT := 16#109300;
        DFCid          : UINT  := 1244;
        debounceMethod : USINT := NATIVE;
    END_STRUCT
END_TYPE

// BODAS_RC18_12_40/Application/02 EasyConfig/DSM_easyConfig/Structure/DFC_MOXEMM_SMU_ALM3_2
{attribute 'external_name' := 'cmp_rts_DFC_MOXEMM_SMU_ALM3_2'}
TYPE DFC_MOXEMM_SMU_ALM3_2 : STRUCT
        DTC            : UDINT := 16#108900;
        DFCid          : UINT  := 1242;
        debounceMethod : USINT := NATIVE;
    END_STRUCT
END_TYPE

// BODAS_RC18_12_40/Application/02 EasyConfig/DSM_easyConfig/Structure/DFC_MOXEMM_SMU_ALM3_4
{attribute 'external_name' := 'cmp_rts_DFC_MOXEMM_SMU_ALM3_4'}
TYPE DFC_MOXEMM_SMU_ALM3_4 : STRUCT
        DTC            : UDINT := 16#108A00;
        DFCid          : UINT  := 1245;
        debounceMethod : USINT := NATIVE;
    END_STRUCT
END_TYPE

// BODAS_RC18_12_40/Application/02 EasyConfig/DSM_easyConfig/Structure/DFC_MOXEMM_SMU_ALM3_5
{attribute 'external_name' := 'cmp_rts_DFC_MOXEMM_SMU_ALM3_5'}
TYPE DFC_MOXEMM_SMU_ALM3_5 : STRUCT
        DTC            : UDINT := 16#108B00;
        DFCid          : UINT  := 1246;
        debounceMethod : USINT := NATIVE;
    END_STRUCT
END_TYPE

// BODAS_RC18_12_40/Application/02 EasyConfig/DSM_easyConfig/Structure/DFC_MOXEMM_SMU_ALM3_7
{attribute 'external_name' := 'cmp_rts_DFC_MOXEMM_SMU_ALM3_7'}
TYPE DFC_MOXEMM_SMU_ALM3_7 : STRUCT
        DTC            : UDINT := 16#108C00;
        DFCid          : UINT  := 1247;
        debounceMethod : USINT := NATIVE;
    END_STRUCT
END_TYPE

// BODAS_RC18_12_40/Application/02 EasyConfig/DSM_easyConfig/Structure/DFC_MOXEMM_SMU_ALM3_8
{attribute 'external_name' := 'cmp_rts_DFC_MOXEMM_SMU_ALM3_8'}
TYPE DFC_MOXEMM_SMU_ALM3_8 : STRUCT
        DTC            : UDINT := 16#108D00;
        DFCid          : UINT  := 1248;
        debounceMethod : USINT := NATIVE;
    END_STRUCT
END_TYPE

// BODAS_RC18_12_40/Application/02 EasyConfig/DSM_easyConfig/Structure/DFC_MOXEMM_SMU_ALM6_0
{attribute 'external_name' := 'cmp_rts_DFC_MOXEMM_SMU_ALM6_0'}
TYPE DFC_MOXEMM_SMU_ALM6_0 : STRUCT
        DTC            : UDINT := 16#109400;
        DFCid          : UINT  := 1249;
        debounceMethod : USINT := NATIVE;
    END_STRUCT
END_TYPE

// BODAS_RC18_12_40/Application/02 EasyConfig/DSM_easyConfig/Structure/DFC_MOXEMM_SMU_ALM6_11
{attribute 'external_name' := 'cmp_rts_DFC_MOXEMM_SMU_ALM6_11'}
TYPE DFC_MOXEMM_SMU_ALM6_11 : STRUCT
        DTC            : UDINT := 16#109900;
        DFCid          : UINT  := 1250;
        debounceMethod : USINT := NATIVE;
    END_STRUCT
END_TYPE

// BODAS_RC18_12_40/Application/02 EasyConfig/DSM_easyConfig/Structure/DFC_MOXEMM_SMU_ALM6_12
{attribute 'external_name' := 'cmp_rts_DFC_MOXEMM_SMU_ALM6_12'}
TYPE DFC_MOXEMM_SMU_ALM6_12 : STRUCT
        DTC            : UDINT := 16#109A00;
        DFCid          : UINT  := 1251;
        debounceMethod : USINT := NATIVE;
    END_STRUCT
END_TYPE

// BODAS_RC18_12_40/Application/02 EasyConfig/DSM_easyConfig/Structure/DFC_MOXEMM_SMU_ALM6_14
{attribute 'external_name' := 'cmp_rts_DFC_MOXEMM_SMU_ALM6_14'}
TYPE DFC_MOXEMM_SMU_ALM6_14 : STRUCT
        DTC            : UDINT := 16#109B00;
        DFCid          : UINT  := 1252;
        debounceMethod : USINT := NATIVE;
    END_STRUCT
END_TYPE

// BODAS_RC18_12_40/Application/02 EasyConfig/DSM_easyConfig/Structure/DFC_MOXEMM_SMU_ALM6_15
{attribute 'external_name' := 'cmp_rts_DFC_MOXEMM_SMU_ALM6_15'}
TYPE DFC_MOXEMM_SMU_ALM6_15 : STRUCT
        DTC            : UDINT := 16#109C00;
        DFCid          : UINT  := 1253;
        debounceMethod : USINT := NATIVE;
    END_STRUCT
END_TYPE

// BODAS_RC18_12_40/Application/02 EasyConfig/DSM_easyConfig/Structure/DFC_MOXEMM_SMU_ALM6_17
{attribute 'external_name' := 'cmp_rts_DFC_MOXEMM_SMU_ALM6_17'}
TYPE DFC_MOXEMM_SMU_ALM6_17 : STRUCT
        DTC            : UDINT := 16#109D00;
        DFCid          : UINT  := 1254;
        debounceMethod : USINT := NATIVE;
    END_STRUCT
END_TYPE

// BODAS_RC18_12_40/Application/02 EasyConfig/DSM_easyConfig/Structure/DFC_MOXEMM_SMU_ALM6_18
{attribute 'external_name' := 'cmp_rts_DFC_MOXEMM_SMU_ALM6_18'}
TYPE DFC_MOXEMM_SMU_ALM6_18 : STRUCT
        DTC            : UDINT := 16#109E00;
        DFCid          : UINT  := 1255;
        debounceMethod : USINT := NATIVE;
    END_STRUCT
END_TYPE

// BODAS_RC18_12_40/Application/02 EasyConfig/DSM_easyConfig/Structure/DFC_MOXEMM_SMU_ALM6_20
{attribute 'external_name' := 'cmp_rts_DFC_MOXEMM_SMU_ALM6_20'}
TYPE DFC_MOXEMM_SMU_ALM6_20 : STRUCT
        DTC            : UDINT := 16#109F00;
        DFCid          : UINT  := 1257;
        debounceMethod : USINT := NATIVE;
    END_STRUCT
END_TYPE

// BODAS_RC18_12_40/Application/02 EasyConfig/DSM_easyConfig/Structure/DFC_MOXEMM_SMU_ALM6_21
{attribute 'external_name' := 'cmp_rts_DFC_MOXEMM_SMU_ALM6_21'}
TYPE DFC_MOXEMM_SMU_ALM6_21 : STRUCT
        DTC            : UDINT := 16#10A000;
        DFCid          : UINT  := 1258;
        debounceMethod : USINT := NATIVE;
    END_STRUCT
END_TYPE

// BODAS_RC18_12_40/Application/02 EasyConfig/DSM_easyConfig/Structure/DFC_MOXEMM_SMU_ALM6_25
{attribute 'external_name' := 'cmp_rts_DFC_MOXEMM_SMU_ALM6_25'}
TYPE DFC_MOXEMM_SMU_ALM6_25 : STRUCT
        DTC            : UDINT := 16#10A100;
        DFCid          : UINT  := 1259;
        debounceMethod : USINT := NATIVE;
    END_STRUCT
END_TYPE

// BODAS_RC18_12_40/Application/02 EasyConfig/DSM_easyConfig/Structure/DFC_MOXEMM_SMU_ALM6_2
{attribute 'external_name' := 'cmp_rts_DFC_MOXEMM_SMU_ALM6_2'}
TYPE DFC_MOXEMM_SMU_ALM6_2 : STRUCT
        DTC            : UDINT := 16#10D900;
        DFCid          : UINT  := 1256;
        debounceMethod : USINT := NATIVE;
    END_STRUCT
END_TYPE

// BODAS_RC18_12_40/Application/02 EasyConfig/DSM_easyConfig/Structure/DFC_MOXEMM_SMU_ALM6_4
{attribute 'external_name' := 'cmp_rts_DFC_MOXEMM_SMU_ALM6_4'}
TYPE DFC_MOXEMM_SMU_ALM6_4 : STRUCT
        DTC            : UDINT := 16#109500;
        DFCid          : UINT  := 1260;
        debounceMethod : USINT := NATIVE;
    END_STRUCT
END_TYPE

// BODAS_RC18_12_40/Application/02 EasyConfig/DSM_easyConfig/Structure/DFC_MOXEMM_SMU_ALM6_5
{attribute 'external_name' := 'cmp_rts_DFC_MOXEMM_SMU_ALM6_5'}
TYPE DFC_MOXEMM_SMU_ALM6_5 : STRUCT
        DTC            : UDINT := 16#109600;
        DFCid          : UINT  := 1261;
        debounceMethod : USINT := NATIVE;
    END_STRUCT
END_TYPE

// BODAS_RC18_12_40/Application/02 EasyConfig/DSM_easyConfig/Structure/DFC_MOXEMM_SMU_ALM6_7
{attribute 'external_name' := 'cmp_rts_DFC_MOXEMM_SMU_ALM6_7'}
TYPE DFC_MOXEMM_SMU_ALM6_7 : STRUCT
        DTC            : UDINT := 16#109700;
        DFCid          : UINT  := 1262;
        debounceMethod : USINT := NATIVE;
    END_STRUCT
END_TYPE

// BODAS_RC18_12_40/Application/02 EasyConfig/DSM_easyConfig/Structure/DFC_MOXEMM_SMU_ALM6_8
{attribute 'external_name' := 'cmp_rts_DFC_MOXEMM_SMU_ALM6_8'}
TYPE DFC_MOXEMM_SMU_ALM6_8 : STRUCT
        DTC            : UDINT := 16#109800;
        DFCid          : UINT  := 1263;
        debounceMethod : USINT := NATIVE;
    END_STRUCT
END_TYPE

// BODAS_RC18_12_40/Application/02 EasyConfig/DSM_easyConfig/Structure/DFC_MOXEMM_SMU_ALM7_12
{attribute 'external_name' := 'cmp_rts_DFC_MOXEMM_SMU_ALM7_12'}
TYPE DFC_MOXEMM_SMU_ALM7_12 : STRUCT
        DTC            : UDINT := 16#10A400;
        DFCid          : UINT  := 1265;
        debounceMethod : USINT := NATIVE;
    END_STRUCT
END_TYPE

// BODAS_RC18_12_40/Application/02 EasyConfig/DSM_easyConfig/Structure/DFC_MOXEMM_SMU_ALM7_13
{attribute 'external_name' := 'cmp_rts_DFC_MOXEMM_SMU_ALM7_13'}
TYPE DFC_MOXEMM_SMU_ALM7_13 : STRUCT
        DTC            : UDINT := 16#10A500;
        DFCid          : UINT  := 1266;
        debounceMethod : USINT := NATIVE;
    END_STRUCT
END_TYPE

// BODAS_RC18_12_40/Application/02 EasyConfig/DSM_easyConfig/Structure/DFC_MOXEMM_SMU_ALM7_14
{attribute 'external_name' := 'cmp_rts_DFC_MOXEMM_SMU_ALM7_14'}
TYPE DFC_MOXEMM_SMU_ALM7_14 : STRUCT
        DTC            : UDINT := 16#10A600;
        DFCid          : UINT  := 1267;
        debounceMethod : USINT := NATIVE;
    END_STRUCT
END_TYPE

// BODAS_RC18_12_40/Application/02 EasyConfig/DSM_easyConfig/Structure/DFC_MOXEMM_SMU_ALM7_15
{attribute 'external_name' := 'cmp_rts_DFC_MOXEMM_SMU_ALM7_15'}
TYPE DFC_MOXEMM_SMU_ALM7_15 : STRUCT
        DTC            : UDINT := 16#10A700;
        DFCid          : UINT  := 1268;
        debounceMethod : USINT := NATIVE;
    END_STRUCT
END_TYPE

// BODAS_RC18_12_40/Application/02 EasyConfig/DSM_easyConfig/Structure/DFC_MOXEMM_SMU_ALM7_16
{attribute 'external_name' := 'cmp_rts_DFC_MOXEMM_SMU_ALM7_16'}
TYPE DFC_MOXEMM_SMU_ALM7_16 : STRUCT
        DTC            : UDINT := 16#10A800;
        DFCid          : UINT  := 1269;
        debounceMethod : USINT := NATIVE;
    END_STRUCT
END_TYPE

// BODAS_RC18_12_40/Application/02 EasyConfig/DSM_easyConfig/Structure/DFC_MOXEMM_SMU_ALM7_17
{attribute 'external_name' := 'cmp_rts_DFC_MOXEMM_SMU_ALM7_17'}
TYPE DFC_MOXEMM_SMU_ALM7_17 : STRUCT
        DTC            : UDINT := 16#10A900;
        DFCid          : UINT  := 1270;
        debounceMethod : USINT := NATIVE;
    END_STRUCT
END_TYPE

// BODAS_RC18_12_40/Application/02 EasyConfig/DSM_easyConfig/Structure/DFC_MOXEMM_SMU_ALM7_1
{attribute 'external_name' := 'cmp_rts_DFC_MOXEMM_SMU_ALM7_1'}
TYPE DFC_MOXEMM_SMU_ALM7_1 : STRUCT
        DTC            : UDINT := 16#10A200;
        DFCid          : UINT  := 1264;
        debounceMethod : USINT := NATIVE;
    END_STRUCT
END_TYPE

// BODAS_RC18_12_40/Application/02 EasyConfig/DSM_easyConfig/Structure/DFC_MOXEMM_SMU_ALM7_20
{attribute 'external_name' := 'cmp_rts_DFC_MOXEMM_SMU_ALM7_20'}
TYPE DFC_MOXEMM_SMU_ALM7_20 : STRUCT
        DTC            : UDINT := 16#10AA00;
        DFCid          : UINT  := 1272;
        debounceMethod : USINT := NATIVE;
    END_STRUCT
END_TYPE

// BODAS_RC18_12_40/Application/02 EasyConfig/DSM_easyConfig/Structure/DFC_MOXEMM_SMU_ALM7_25
{attribute 'external_name' := 'cmp_rts_DFC_MOXEMM_SMU_ALM7_25'}
TYPE DFC_MOXEMM_SMU_ALM7_25 : STRUCT
        DTC            : UDINT := 16#10AB00;
        DFCid          : UINT  := 1273;
        debounceMethod : USINT := NATIVE;
    END_STRUCT
END_TYPE

// BODAS_RC18_12_40/Application/02 EasyConfig/DSM_easyConfig/Structure/DFC_MOXEMM_SMU_ALM7_26
{attribute 'external_name' := 'cmp_rts_DFC_MOXEMM_SMU_ALM7_26'}
TYPE DFC_MOXEMM_SMU_ALM7_26 : STRUCT
        DTC            : UDINT := 16#10AC00;
        DFCid          : UINT  := 1274;
        debounceMethod : USINT := NATIVE;
    END_STRUCT
END_TYPE

// BODAS_RC18_12_40/Application/02 EasyConfig/DSM_easyConfig/Structure/DFC_MOXEMM_SMU_ALM7_28
{attribute 'external_name' := 'cmp_rts_DFC_MOXEMM_SMU_ALM7_28'}
TYPE DFC_MOXEMM_SMU_ALM7_28 : STRUCT
        DTC            : UDINT := 16#10AD00;
        DFCid          : UINT  := 1275;
        debounceMethod : USINT := NATIVE;
    END_STRUCT
END_TYPE

// BODAS_RC18_12_40/Application/02 EasyConfig/DSM_easyConfig/Structure/DFC_MOXEMM_SMU_ALM7_29
{attribute 'external_name' := 'cmp_rts_DFC_MOXEMM_SMU_ALM7_29'}
TYPE DFC_MOXEMM_SMU_ALM7_29 : STRUCT
        DTC            : UDINT := 16#10AE00;
        DFCid          : UINT  := 1276;
        debounceMethod : USINT := NATIVE;
    END_STRUCT
END_TYPE

// BODAS_RC18_12_40/Application/02 EasyConfig/DSM_easyConfig/Structure/DFC_MOXEMM_SMU_ALM7_2
{attribute 'external_name' := 'cmp_rts_DFC_MOXEMM_SMU_ALM7_2'}
TYPE DFC_MOXEMM_SMU_ALM7_2 : STRUCT
        DTC            : UDINT := 16#10A300;
        DFCid          : UINT  := 1271;
        debounceMethod : USINT := NATIVE;
    END_STRUCT
END_TYPE

// BODAS_RC18_12_40/Application/02 EasyConfig/DSM_easyConfig/Structure/DFC_MOXEMM_SMU_ALM7_30
{attribute 'external_name' := 'cmp_rts_DFC_MOXEMM_SMU_ALM7_30'}
TYPE DFC_MOXEMM_SMU_ALM7_30 : STRUCT
        DTC            : UDINT := 16#10AF00;
        DFCid          : UINT  := 1277;
        debounceMethod : USINT := NATIVE;
    END_STRUCT
END_TYPE

// BODAS_RC18_12_40/Application/02 EasyConfig/DSM_easyConfig/Structure/DFC_MOXEMM_SMU_ALM7_31
{attribute 'external_name' := 'cmp_rts_DFC_MOXEMM_SMU_ALM7_31'}
TYPE DFC_MOXEMM_SMU_ALM7_31 : STRUCT
        DTC            : UDINT := 16#10B000;
        DFCid          : UINT  := 1278;
        debounceMethod : USINT := NATIVE;
    END_STRUCT
END_TYPE

// BODAS_RC18_12_40/Application/02 EasyConfig/DSM_easyConfig/Structure/DFC_MOXEMM_SMU_ALM8_0
{attribute 'external_name' := 'cmp_rts_DFC_MOXEMM_SMU_ALM8_0'}
TYPE DFC_MOXEMM_SMU_ALM8_0 : STRUCT
        DTC            : UDINT := 16#10B100;
        DFCid          : UINT  := 1279;
        debounceMethod : USINT := NATIVE;
    END_STRUCT
END_TYPE

// BODAS_RC18_12_40/Application/02 EasyConfig/DSM_easyConfig/Structure/DFC_MOXEMM_SMU_ALM8_10
{attribute 'external_name' := 'cmp_rts_DFC_MOXEMM_SMU_ALM8_10'}
TYPE DFC_MOXEMM_SMU_ALM8_10 : STRUCT
        DTC            : UDINT := 16#10B600;
        DFCid          : UINT  := 1281;
        debounceMethod : USINT := NATIVE;
    END_STRUCT
END_TYPE

// BODAS_RC18_12_40/Application/02 EasyConfig/DSM_easyConfig/Structure/DFC_MOXEMM_SMU_ALM8_11
{attribute 'external_name' := 'cmp_rts_DFC_MOXEMM_SMU_ALM8_11'}
TYPE DFC_MOXEMM_SMU_ALM8_11 : STRUCT
        DTC            : UDINT := 16#10B700;
        DFCid          : UINT  := 1282;
        debounceMethod : USINT := NATIVE;
    END_STRUCT
END_TYPE

// BODAS_RC18_12_40/Application/02 EasyConfig/DSM_easyConfig/Structure/DFC_MOXEMM_SMU_ALM8_12
{attribute 'external_name' := 'cmp_rts_DFC_MOXEMM_SMU_ALM8_12'}
TYPE DFC_MOXEMM_SMU_ALM8_12 : STRUCT
        DTC            : UDINT := 16#10B800;
        DFCid          : UINT  := 1283;
        debounceMethod : USINT := NATIVE;
    END_STRUCT
END_TYPE

// BODAS_RC18_12_40/Application/02 EasyConfig/DSM_easyConfig/Structure/DFC_MOXEMM_SMU_ALM8_13
{attribute 'external_name' := 'cmp_rts_DFC_MOXEMM_SMU_ALM8_13'}
TYPE DFC_MOXEMM_SMU_ALM8_13 : STRUCT
        DTC            : UDINT := 16#10B900;
        DFCid          : UINT  := 1284;
        debounceMethod : USINT := NATIVE;
    END_STRUCT
END_TYPE

// BODAS_RC18_12_40/Application/02 EasyConfig/DSM_easyConfig/Structure/DFC_MOXEMM_SMU_ALM8_16
{attribute 'external_name' := 'cmp_rts_DFC_MOXEMM_SMU_ALM8_16'}
TYPE DFC_MOXEMM_SMU_ALM8_16 : STRUCT
        DTC            : UDINT := 16#10BA00;
        DFCid          : UINT  := 1285;
        debounceMethod : USINT := NATIVE;
    END_STRUCT
END_TYPE

// BODAS_RC18_12_40/Application/02 EasyConfig/DSM_easyConfig/Structure/DFC_MOXEMM_SMU_ALM8_18
{attribute 'external_name' := 'cmp_rts_DFC_MOXEMM_SMU_ALM8_18'}
TYPE DFC_MOXEMM_SMU_ALM8_18 : STRUCT
        DTC            : UDINT := 16#10BB00;
        DFCid          : UINT  := 1286;
        debounceMethod : USINT := NATIVE;
    END_STRUCT
END_TYPE

// BODAS_RC18_12_40/Application/02 EasyConfig/DSM_easyConfig/Structure/DFC_MOXEMM_SMU_ALM8_1
{attribute 'external_name' := 'cmp_rts_DFC_MOXEMM_SMU_ALM8_1'}
TYPE DFC_MOXEMM_SMU_ALM8_1 : STRUCT
        DTC            : UDINT := 16#10B200;
        DFCid          : UINT  := 1280;
        debounceMethod : USINT := NATIVE;
    END_STRUCT
END_TYPE

// BODAS_RC18_12_40/Application/02 EasyConfig/DSM_easyConfig/Structure/DFC_MOXEMM_SMU_ALM8_2
{attribute 'external_name' := 'cmp_rts_DFC_MOXEMM_SMU_ALM8_2'}
TYPE DFC_MOXEMM_SMU_ALM8_2 : STRUCT
        DTC            : UDINT := 16#10B300;
        DFCid          : UINT  := 1287;
        debounceMethod : USINT := NATIVE;
    END_STRUCT
END_TYPE

// BODAS_RC18_12_40/Application/02 EasyConfig/DSM_easyConfig/Structure/DFC_MOXEMM_SMU_ALM8_30
{attribute 'external_name' := 'cmp_rts_DFC_MOXEMM_SMU_ALM8_30'}
TYPE DFC_MOXEMM_SMU_ALM8_30 : STRUCT
        DTC            : UDINT := 16#10BC00;
        DFCid          : UINT  := 1289;
        debounceMethod : USINT := NATIVE;
    END_STRUCT
END_TYPE

// BODAS_RC18_12_40/Application/02 EasyConfig/DSM_easyConfig/Structure/DFC_MOXEMM_SMU_ALM8_31
{attribute 'external_name' := 'cmp_rts_DFC_MOXEMM_SMU_ALM8_31'}
TYPE DFC_MOXEMM_SMU_ALM8_31 : STRUCT
        DTC            : UDINT := 16#10BD00;
        DFCid          : UINT  := 1290;
        debounceMethod : USINT := NATIVE;
    END_STRUCT
END_TYPE

// BODAS_RC18_12_40/Application/02 EasyConfig/DSM_easyConfig/Structure/DFC_MOXEMM_SMU_ALM8_3
{attribute 'external_name' := 'cmp_rts_DFC_MOXEMM_SMU_ALM8_3'}
TYPE DFC_MOXEMM_SMU_ALM8_3 : STRUCT
        DTC            : UDINT := 16#10B400;
        DFCid          : UINT  := 1288;
        debounceMethod : USINT := NATIVE;
    END_STRUCT
END_TYPE

// BODAS_RC18_12_40/Application/02 EasyConfig/DSM_easyConfig/Structure/DFC_MOXEMM_SMU_ALM8_4
{attribute 'external_name' := 'cmp_rts_DFC_MOXEMM_SMU_ALM8_4'}
TYPE DFC_MOXEMM_SMU_ALM8_4 : STRUCT
        DTC            : UDINT := 16#10B500;
        DFCid          : UINT  := 1291;
        debounceMethod : USINT := NATIVE;
    END_STRUCT
END_TYPE

// BODAS_RC18_12_40/Application/02 EasyConfig/DSM_easyConfig/Structure/DFC_MOXEMM_SMU_ALM9_0
{attribute 'external_name' := 'cmp_rts_DFC_MOXEMM_SMU_ALM9_0'}
TYPE DFC_MOXEMM_SMU_ALM9_0 : STRUCT
        DTC            : UDINT := 16#10BE00;
        DFCid          : UINT  := 1292;
        debounceMethod : USINT := NATIVE;
    END_STRUCT
END_TYPE

// BODAS_RC18_12_40/Application/02 EasyConfig/DSM_easyConfig/Structure/DFC_MOXEMM_SMU_ALM9_15
{attribute 'external_name' := 'cmp_rts_DFC_MOXEMM_SMU_ALM9_15'}
TYPE DFC_MOXEMM_SMU_ALM9_15 : STRUCT
        DTC            : UDINT := 16#10C100;
        DFCid          : UINT  := 1294;
        debounceMethod : USINT := NATIVE;
    END_STRUCT
END_TYPE

// BODAS_RC18_12_40/Application/02 EasyConfig/DSM_easyConfig/Structure/DFC_MOXEMM_SMU_ALM9_1
{attribute 'external_name' := 'cmp_rts_DFC_MOXEMM_SMU_ALM9_1'}
TYPE DFC_MOXEMM_SMU_ALM9_1 : STRUCT
        DTC            : UDINT := 16#10BF00;
        DFCid          : UINT  := 1293;
        debounceMethod : USINT := NATIVE;
    END_STRUCT
END_TYPE

// BODAS_RC18_12_40/Application/02 EasyConfig/DSM_easyConfig/Structure/DFC_MOXEMM_SMU_ALM9_3
{attribute 'external_name' := 'cmp_rts_DFC_MOXEMM_SMU_ALM9_3'}
TYPE DFC_MOXEMM_SMU_ALM9_3 : STRUCT
        DTC            : UDINT := 16#10C000;
        DFCid          : UINT  := 1295;
        debounceMethod : USINT := NATIVE;
    END_STRUCT
END_TYPE

// BODAS_RC18_12_40/Application/02 EasyConfig/DSM_easyConfig/Structure/DFC_MoXEMMHwLTLBIST
{attribute 'external_name' := 'cmp_rts_DFC_MoXEMMHwLTLBIST'}
TYPE DFC_MoXEMMHwLTLBIST : STRUCT
        DTC : UDINT := 16#10D000;
    END_STRUCT
END_TYPE

// BODAS_RC18_12_40/Application/02 EasyConfig/DSM_easyConfig/Structure/DFC_MoXEMMHwLTMBIST
{attribute 'external_name' := 'cmp_rts_DFC_MoXEMMHwLTMBIST'}
TYPE DFC_MoXEMMHwLTMBIST : STRUCT
        DTC : UDINT := 16#10D100;
    END_STRUCT
END_TYPE

// BODAS_RC18_12_40/Application/02 EasyConfig/DSM_easyConfig/Structure/DFC_MoXEMMHwLTMCUFW
{attribute 'external_name' := 'cmp_rts_DFC_MoXEMMHwLTMCUFW'}
TYPE DFC_MoXEMMHwLTMCUFW : STRUCT
        DTC            : UDINT := 16#10D200;
        DFCid          : UINT  := 1299;
        debounceMethod : USINT := NATIVE;
    END_STRUCT
END_TYPE

// BODAS_RC18_12_40/Application/02 EasyConfig/DSM_easyConfig/Structure/DFC_MoXEMMHwLTMonBIST
{attribute 'external_name' := 'cmp_rts_DFC_MoXEMMHwLTMonBIST'}
TYPE DFC_MoXEMMHwLTMonBIST : STRUCT
        DTC            : UDINT := 16#10D300;
        DFCid          : UINT  := 1300;
        debounceMethod : USINT := NATIVE;
    END_STRUCT
END_TYPE

// BODAS_RC18_12_40/Application/02 EasyConfig/DSM_easyConfig/Structure/DFC_MoXEMMHwLTRegMonTest
{attribute 'external_name' := 'cmp_rts_DFC_MoXEMMHwLTRegMonTest'}
TYPE DFC_MoXEMMHwLTRegMonTest : STRUCT
        DTC            : UDINT := 16#10D400;
        DFCid          : UINT  := 1301;
        debounceMethod : USINT := NATIVE;
    END_STRUCT
END_TYPE

// BODAS_RC18_12_40/Application/02 EasyConfig/DSM_easyConfig/Structure/DFC_MoXEMMHwLTStbySMUAlvTest
{attribute 'external_name' := 'cmp_rts_DFC_MoXEMMHwLTStbySMUAlvTest'}
TYPE DFC_MoXEMMHwLTStbySMUAlvTest : STRUCT
        DTC            : UDINT := 16#10D500;
        DFCid          : UINT  := 1302;
        debounceMethod : USINT := NATIVE;
    END_STRUCT
END_TYPE

// BODAS_RC18_12_40/Application/GlobalVariables
VAR_GLOBAL
    PrmAsw_gstruc             : struc_para;
    anValue_perc_gu8          : USINT;
    swtStatus_gu8             : USINT;
    can1RxDataboxCbkCntr_gu32 : UDINT;
END_VAR
VAR_GLOBAL CONSTANT
    PrmAsw_cgstruc : struc_para := (fctPmp_s16       := 0,
                                    listCtrlVlv_enu  := 1,
                                    nrCogs_s16       := 33,
                                    iSpSafout1_u16   := 500,
                                    iSpSafout2_u16   := 500,
                                    eff_perc_au16    := [10, 50, 90],
                                    nEngSpd_rpm_au16 := [500, 2000, 3500],
                                    PrmDbg_struc     := (flgXcpOn_b := FALSE, flgStoreDataToNvm_b := FALSE));
    ErrMemMgr_nrDfesEntries_DU8 : USINT := 32; (* Maximum number OF errors in DFES *)
    ErrMemMgr_stNoEntryAvl_DU8  : USINT := 255;
    (* bit masks for error states *)
    ErrMemMgr_BitMaskErrDeactvNotSave_DU8 : BYTE := 16#01; (* mask TO fetch Deactive errors which are NOT saved yet *)
    ErrMemMgr_BitMaskErrPrevActv_DU8      : BYTE := 16#10; (* mask TO fetch previously active errors *)
    ErrMemMgr_BitMaskErrActv_DU8          : BYTE := 16#03; (* mask TO fetch active errors *)
    ErrMemMgr_BitMaskErrDeactvSaved_DU8   : BYTE := 16#04; (* mask TO fetch saved deactive errors *)
    ErrMemMgr_BitMaskErrSts_DU8           : BYTE := 16#FF; (* default mask *)
    ErrMemMgr_nrMaxErrEntry_DU8           : BYTE := 27;    (* Max. number of entries, before deleting starts *)
END_VAR

// BODAS_RC18_12_40/Application/02 EasyConfig/Lin_CanSignals_easyConfig/GVL_linCanSignals_easyConfig
VAR_GLOBAL
    PDUR_VARIANT_PRE_COMPILE                                    : USINT := 0;
    PDUR_VARIANT_POSTBUILD_LOADABLE                             : USINT := 1;
    PDUR_CONFIGURATION_VARIANT                                  : USINT := PDUR_VARIANT_PRE_COMPILE;
    PduRConf_PduRSrcPdu_CddToPduR_HWVrsNumIBS2105_Src           : USINT := 0;
    PduRConf_PduRDestPdu_PduRToLinTp_HWVrsNumIBS2105_Dest       : USINT := 0;
    PduRConf_PduRSrcPdu_DoIP_Rx_DoIP2PduR_Src_Java              : USINT := 0;
    PduRConf_PduRDestPdu_DoIP_Rx_PduR2Dcm_Dest_Java             : USINT := 0;
    PduRConf_PduRSrcPdu_DoIP_Tx_Dcm2PduR_Src_JavaTool           : USINT := 0;
    PduRConf_PduRDestPdu_DoIP_Tx_PduR2DoIP_Dest_Java            : USINT := 0;
    PduRConf_PduRSrcPdu_LinTPToPduR_HWVrsNumIBS2105_Src         : USINT := 0;
    PduRConf_PduRDestPdu_PduRToCdd_HWVrsNumIBS2105_Dest         : USINT := 0;
    PduRConf_PduRSrcPdu_NM_TX_FA_Com2PduR_Src                   : USINT := 0;
    PduRConf_PduRDestPdu_NM_TX_FA_PduR2CanNm_Dest               : USINT := 0;
    PduRConf_PduRSrcPdu_rbr_Pdu_Com2PduR_CCVS_xTx_Src           : USINT := 1;
    PduRConf_PduRDestPdu_rbr_Pdu_CanIf_CCVS_xTx_Dest            : USINT := 0;
    PduRConf_PduRSrcPdu_rbr_Pdu_CanIf_sig_C_xRx_Src             : USINT := 1;
    PduRConf_PduRSrcPdu_rbr_Pdu_Com2PduR_C_xTx_Src              : USINT := 2;
    PduRConf_PduRDestPdu_rbr_Pdu_CanIf_sig_C_xTx_Dest           : USINT := 1;
    PduRConf_PduRSrcPdu_rbr_Pdu_CanIf_EngCtrl1_xRx_Dest         : USINT := 0;
    PduRConf_PduRSrcPdu_UdsOnCan_FctExtdidRx_CanTp2PduR_Src     : USINT := 0;
    PduRConf_PduRDestPdu_UdsOnCan_FctExtdidRx_PduR2Dcm_Dest     : USINT := 1;
    PduRConf_PduRSrcPdu_UdsOnCan_PhyRxExtdId_CanTp2PduR_Src     : USINT := 1;
    PduRConf_PduRDestPdu_UdsOnCan_PhyRxExtdId_PduR2Dcm_Dest     : USINT := 2;
    PduRConf_PduRSrcPdu_UdsOnCan_PhyTxExtdId_Dcm2PduR_Src       : USINT := 1;
    PduRConf_PduRDestPdu_UdsOnCan_PhyTxExtdId_PduR2CanTp_Dest   : USINT := 0;
    LinIfConf_LinIfChannel_LinIfChannel_0                       : USINT := 5;
    LinIfConf_LinIfFrame_LinIf_MRF                              : USINT := 16#00;
    LinIfConf_LinIfFrame_LinIf_SRF                              : USINT := 16#01;
    NULL_SCHEDULE                                               : USINT := 16#00;
    LinIf_Scht_MasterReq_LinIfChannel_0_bds_Pb_preDefRef_vrnt01 : USINT := 16#01;
    LinIf_Scht_SlaveResp_LinIfChannel_0_bds_Pb_preDefRef_vrnt01 : USINT := 16#02;
    LinIf_Scht_RUN_MAIN_LinIfChannel_0_bds_Pb_preDefRef_vrnt01  : USINT := 16#03;
    COM_VARIANT_PRE_COMPILE                                     : USINT := 0;
    COM_VARIANT_LINK_TIME                                       : USINT := 1;
    COM_VARIANT_POSTBUILD_LOADABLE                              : USINT := 2;
    COM_VARIANT_POSTBUILD_SELECTABLE                            : USINT := 3;
    COM_CONFIGURATION_VARIANT                                   : USINT := COM_VARIANT_PRE_COMPILE;
    ComConf_ComIPdu_ComIPdu_CCVS_xTx                            : USINT := 0;
    ComConf_ComIPdu_ComIPdu_C_xTx                               : USINT := 1;
    ComConf_ComIPdu_NM_TX_FA                                    : USINT := 2;
    ComConf_ComIPdu_ComIPdu_C_xRx                               : USINT := 0;
    ComConf_ComIPdu_ComIPdu_EngCtrl1_xRx                        : USINT := 1;
    ComConf_ComSignal_ComSignal_WheelBasedVehicleSpeed_xTx      : USINT := 0;
    ComConf_ComSignal_ComSignal_ParkingBrakeSwitch_xTx          : USINT := 1;
    ComConf_ComSignal_ComSignal_C_xTx                           : USINT := 2;
    ComConf_ComSignal_ComSignal_C_xRx                           : USINT := 0;
    ComConf_ComSignal_ComSignal_EngSpeed_xRx                    : USINT := 1;
    ComConf_ComSignal_ComSignal_ActualEngPercentTorque_xRx      : USINT := 2;
    ComConf_ComSignalGroup_ComSignalGroup_Tx_1                  : USINT := 0;
    ComConf_ComSignalGroup_ComSignalGroup_Rx_1                  : USINT := 0;
    ComConf_ComGroupSignal_ComGroupSignal_Tx                    : USINT := 0;
    ComConf_ComGroupSignal_ComGroupSignal_Rx                    : USINT := 0;
    ComConf_ComIPduGroup_ComIPduGroup_CAN_2_Rx                  : USINT := 0;
    ComConf_ComIPduGroup_ComIPduGroup_CAN_2_Tx                  : USINT := 1;
    ComConf_ComIPduGroup_ComIPduGroup_C_Rx                      : USINT := 2;
    ComConf_ComIPduGroup_ComIPduGroup_C_Tx                      : USINT := 3;
    ComConf_ComIPduGroup_LE_CAN_NM_TX                           : USINT := 4;
    ComConf_ComIPduGroup_LP_CAN_NM_TX                           : USINT := 5;
    ComConf_ComIPduGroup_LinChannel_0_RX                        : USINT := 6;
    ComConf_ComIPduGroup_LinChannel_0_TX                        : USINT := 7;
    ComConf_ComIPduGroup_LinRx                                  : USINT := 8;
    ComConf_ComIPduGroup_LinTx                                  : USINT := 9;
    ComConf_ComIPduGroup_MLIN_RX                                : USINT := 10;
    ComConf_ComIPduGroup_MLIN_TX                                : USINT := 11;
    ComConf_ComIPduGroup_PT_CAN_RX                              : USINT := 12;
    ComConf_ComIPduGroup_PT_CAN_TX                              : USINT := 13;
    BDS_LIN_CHNL_1_DU8                                          : USINT := LinIfConf_LinIfChannel_LinIfChannel_0;
END_VAR

// BODAS_RC18_12_40/Application/02 EasyConfig/DSM_easyConfig/GVL/GVL_debounceMethod
VAR_GLOBAL
    TIME_IN_ROW         : USINT := 0;
    EVENT_IN_ROW        : USINT := 1;
    TIME_UP_DOWN        : USINT := 2;
    EVENT_UP_DOWN       : USINT := 3;
    TIME_UP_DOWN_SMALL  : USINT := 4;
    EVENT_UP_DOWN_SMALL : USINT := 5;
    TIME_IN_ROW_SMALL   : USINT := 6;
    EVENT_IN_ROW_SMALL  : USINT := 7;
    NO_DEBOUNCE         : USINT := 8;
    NATIVE              : USINT := 8;
END_VAR

// BODAS_RC18_12_40/Application/MAIN_TASK_PRG
(*********************************************************************************************************************
 *    __   __   ___  ___           __   __        __   __  ___
 *   /_ / /  / /__  /    /__/     /_ / /_   |_ / /_ / /  /  /  /__/
 *  /__/ /__/ __ / /__  /  /     /  | /__  /  | /  | /__/  /  /  /
 *
 * Project: Hello World for ml290.rts
 *
 * Program: Main_Task_PRG
 *
 * Description:
 * Main loop of application
 *
 * (c) Copyright by BOSCH REXROTH AG, all rights reserved
 *
 *********************************************************************************************************************)
PROGRAM MAIN_TASK_PRG
VAR
    (******************************************************************************)
    (*************************** _Init ********************************************)
    (******************************************************************************)
    (******************************************************************************)
    (*************************** _Starlock ****************************************)
    (******************************************************************************)
    StartRelease_st_b : BOOL; (*State of the startlock: 1 = the program runs*)
    (******************************************************************************)
    (*************************** _Run *********************************************)
    (******************************************************************************)
    (******************************************************************************)
    (*************************** _PostRun *****************************************)
    (******************************************************************************)
    PostRun_st_b         : BOOL; (*State of the postrun: 1 = the post runs*)
    CallPostRunNr_no_u16 : UINT;
    States_s             : bds_sys_states_ts;
    (******************************************************************************)
    (*************************** _Errors ******************************************)
    (******************************************************************************)
    (******************************************************************************)
    (*************************** _CAN *********************************************)
    (******************************************************************************)
    (******************************************************************************)
    (*************************** General ******************************************)
    (******************************************************************************)
    st_Startlock_b    : BOOL;
    MainTaskState_enu : enu_MainTaskState :=
        enu_MainTaskState.MT_INIT; (* variable indicating the mode of the main task callback function (MT_INIT, MT_CYCLE) *)
END_VAR
VAR CONSTANT
    DELAY_STANDARD       : INT  := 2000; (* debouncing time 2000[ms]*)
    TaskCycleTime_ms_u16 : UINT := 10;   (* Task Cycle Time *)
END_VAR

CASE MainTaskState_enu OF
enu_MainTaskState.MT_INIT:
    (* Initialization state - only once *)
    INIT();
    StartRelease_st_b := FALSE;
    MainTaskState_enu := enu_MainTaskState.MT_CYCLE;
    ELSE (* -> MT_CYCLE and default state *)
        (* Cyclic state *)
        (* Read inputs *)
        INPUTS();

        IF (StartRelease_st_b) THEN
            IF (PostRun_st_b) THEN
                (* Postrun *)
                POSTRUN();
            ELSE
                (* Normal operational mode *)
                //_RUN();
            END_IF
        ELSE
            (* Wait for start release *)
            STARTLOCK();
        END_IF

        (* Set CAN outputs *)
        CAN_OUT();
        (* Error management *)
        ERRORS();
        (* Set outputs *)
        OUTPUTS();
        (* Reads the parameter from EEPROM *)
        READ_PARAMETERS();
END_CASE

ACTION CAN_OUT:
(******************************************************************************)
(******************** CAN OUTPUT  *********************************************)
(******************************************************************************)
PRG_CANOut(i_statusNvmIni_u16  := PRG_NVMConfig.status_u16,
           i_iPmpFwdAct_mA_u16 := PRG_Outputs.no_CurrentK07_mA_u16,
           i_iPmpFwdSet_mA_u16 := PRG_Outputs.iPmpFwdSet_mA_u16,
           i_CtrlValve_u8      := PRG_Outputs.st_CtrlValve_u8,
           i_rxActEngPercTq_u8 := PRG_CANIn.o_rxActEngPercTq_u8,
           i_vWhlSpd_kph_u16   := UINT_TO_INT(PRG_Inputs.vWhlSpd_kph_u16),
           i_uPmpSnsr_mV_u16   := PRG_Inputs.uPmpSnsr_mV_u16,
           i_frqVehSnsr_Hz_u32 := PRG_Inputs.frqVehSnsr_Hz_u32,
           i_anValue_perc_u8   := GlobalVariables.anValue_perc_gu8,
           i_stBrkSwt_u8       := PRG_Outputs.st_BrkSwt_u8);
END_ACTION

ACTION ERRORS:
(******************************************************************************)
(******************** Error Handling  *****************************************)
(******************************************************************************)
PRG_HandleErrors(i_stPmpSnsrSigInvldErr_e := PRG_Inputs.stPmpSnsrSigInvldErr_e,
                 i_stBrkSwtSigInvldErr_e  := PRG_Inputs.stBrkSwtSigInvldErr_e,
                 i_uPmpSnsr_mV_u16        := PRG_Inputs.uPmpSnsr_mV_u16,
                 i_frqVehSnsr_Hz_u32      := UDINT_TO_UINT(PRG_Inputs.frqVehSnsr_Hz_u32),
                 i_iPmpFwdAct_mA_u16      := PRG_Outputs.no_CurrentK07_mA_u16,
                 i_vWhlSpd_kmh_u16        := PRG_Inputs.vWhlSpd_kph_u16);

(******************************************************************************)
(******************** Error Memory Workaround *********************************)
(******************************************************************************)
PRG_ErrMemMgr();
END_ACTION

ACTION INIT:
(******************************************************************************)
(******************** INIT  ***************************************************)
(******************************************************************************)
INIT_PRG();
END_ACTION

ACTION INPUTS:
(******************************************************************************)
(************************ INPUTS  *********************************************)
(******************************************************************************)
PRG_Inputs(i_TaskCycleTime_ms_u16 := TaskCycleTime_ms_u16, o_T15_st_u8 =>);
(******************************************************************************)
(************************ CAN INPUT  ******************************************)
(******************************************************************************)
PRG_CANIn();
(* read current and previous states of system. *)
bds_sys_getStates(ADR(states_s));

(* if the system is in POSTRUN state currently *)
IF (NOT (USINT_TO_BOOL(PRG_Inputs.o_T15_st_u8)) OR states_s.currentState_e = BDS_SYSSTATE_POSTRUN_E) THEN
    PostRun_st_b := TRUE;
ELSE
    PostRun_st_b := FALSE;
END_IF
END_ACTION

ACTION OUTPUTS:
(******************************************************************************)
(************************ OUTPUTS  ********************************************)
(******************************************************************************)
PRG_Outputs(i_UPumpSensr_mV_u16 := PRG_Inputs.uPmpSnsr_mV_u16);
END_ACTION

